# B&R Automation Studio project NAELD004C00R10L518F00 (part 6)

#### Act_Main_P1021.st
```iecst
ACTION Act_Main_P1021:

	//Machine Setting - General
	tyP1021McSetGen.tyGen.tyNumConvInitTm.diValueMin	:= p_tyNtParamCurr.tyUIConvInitTm.diMin;
	tyP1021McSetGen.tyGen.tyNumConvInitTm.diValueMax	:= p_tyNtParamCurr.tyUIConvInitTm.diMax;

	tyP1021McSetGen.tyGen.tyNumMag1ConvRunTm.diValueMin	:= p_tyNtParamCurr.tyUIMagConvRunTm.diMin;
	tyP1021McSetGen.tyGen.tyNumMag1ConvRunTm.diValueMax	:= p_tyNtParamCurr.tyUIMagConvRunTm.diMax;
	tyP1021McSetGen.tyGen.tyNumMag2ConvRunTm.diValueMin	:= p_tyNtParamCurr.tyUIMagConvRunTm.diMin;
	tyP1021McSetGen.tyGen.tyNumMag2ConvRunTm.diValueMax	:= p_tyNtParamCurr.tyUIMagConvRunTm.diMax;
	tyP1021McSetGen.tyGen.tyNumMag3ConvRunTm.diValueMin	:= p_tyNtParamCurr.tyUIMagConvRunTm.diMin;
	tyP1021McSetGen.tyGen.tyNumMag3ConvRunTm.diValueMax	:= p_tyNtParamCurr.tyUIMagConvRunTm.diMax;
	tyP1021McSetGen.tyGen.tyNumMag4ConvRunTm.diValueMin	:= p_tyNtParamCurr.tyUIMagConvRunTm.diMin;
	tyP1021McSetGen.tyGen.tyNumMag4ConvRunTm.diValueMax	:= p_tyNtParamCurr.tyUIMagConvRunTm.diMax;

	tyP1021McSetGen.tyGen.tyNumTranOutErrDlyTm.diValueMin	:= p_tyNtParamCurr.tyUITranOutErrDlyTm.diMin;
	tyP1021McSetGen.tyGen.tyNumTranOutErrDlyTm.diValueMax	:= p_tyNtParamCurr.tyUITranOutErrDlyTm.diMax;

	//LMC feedback time
	tyP1021McSetGen.tyGen.tyNumLMCFbTm.uiRtStat	:= NOT p_tyNtParamCurr.bProjWorkOrderOPCUA;

	//Screen Saver
	tyP1021McSetGen.tyGen.tyNumSSaverTm.diValueMin	:= p_tyNtParamCurr.tyUISSaverTm.diMin;
	tyP1021McSetGen.tyGen.tyNumSSaverTm.diValueMax	:= p_tyNtParamCurr.tyUISSaverTm.diMax;
	tyP1021McSetGen.tyGen.tyNumSSaverTm.uiRtStat.0	:= NOT p_tyNtParamCurr.bSSaverPrep;
	tyP1021McSetGen.tyGen.tyBtnSSaverEn.uiRtStat.0	:= NOT p_tyNtParamCurr.bSSaverPrep;
	tyP1021McSetGen.tyGen.tyTxtLblSSaver.uiRtStat.0	:= NOT p_tyNtParamCurr.bSSaverPrep;

	//Width
	tyP1021McSetGen.tyGen.tyNumWidthAtHm.diValueMin	:= p_tyNtParamCurr.tyProdRcpWidth.diMin;
	tyP1021McSetGen.tyGen.tyNumWidthAtHm.diValueMax	:= p_tyNtParamCurr.tyProdRcpWidth.diMax + 10000;
	tyP1021McSetGen.tyGen.tyNumWidthAtHm.uiRtStat.0	:= NOT p_tyNtParamCurr.bAWPrep;
	tyP1021McSetGen.tyGen.tyTxtWidthAtHm.uiRtStat.0	:= NOT p_tyNtParamCurr.bAWPrep;
	tyP1021McSetGen.tyGen.tyBtnAWDis.uiRtStat.0		:= NOT p_tyNtParamCurr.bAWPrep;

	//Pusher Auto Width AT Home
	tyP1021McSetGen.tyGen.tyNumAWPusherAtHm.diValueMin	:= p_tyNtParamCurr.tyProdRcpWidth.diMin-p_tyNtParamCurr.tyProdRcpWidth.diMin;
	tyP1021McSetGen.tyGen.tyNumAWPusherAtHm.diValueMax	:= (p_tyNtParamCurr.tyProdRcpWidth.diMax + 10000) / 2;
	tyP1021McSetGen.tyGen.tyNumAWPusherAtHm.uiRtStat.0	:= NOT p_tyNtParamCurr.bAWPusherPrep;
	tyP1021McSetGen.tyGen.tyTxtAWPusherAtHm.uiRtStat.0	:= NOT p_tyNtParamCurr.bAWPusherPrep;
	tyP1021McSetGen.tyGen.tyBtnAWPusherDis.uiRtStat.0	:= NOT p_tyNtParamCurr.bAWPusherPrep;

//	tyP1021McSetGen.tyGen.tyNumWidthOffset.uiRtStat.0 :=  NOT p_tyNtParamCurr.bAWPrep;
//	tyP1021McSetGen.tyGen.tyTxtWidthOffset.uiRtStat.0 :=  NOT p_tyNtParamCurr.bAWPrep;
	tyP1021McSetGen.tyGen.tyNumWidthOffset.uiRtStat.0 := TRUE;
	tyP1021McSetGen.tyGen.tyTxtWidthOffset.uiRtStat.0 := TRUE;
	tyP1021McSetGen.tyGen.tyNumWidthOffset.diValueMin :=  p_tyNtParamCurr.tyUIAWOffset.diMin;
	tyP1021McSetGen.tyGen.tyNumWidthOffset.diValueMax :=  p_tyNtParamCurr.tyUIAWOffset.diMax;
	//Hermes Remote Configuration
	tyP1021McSetGen.tyGen.tyBtnHermesRmtEn.uiRtStat.0	:= NOT p_tyNtParamCurr.bHermesRmtPrep;

	//Machine Mode
	tyP1021McSetGen.tyGen.tyDrpDnDefaultMcMod.uiRtStat.0 := TRUE;
	IF p_tyNtParamCurr.bProjLaneBPrep THEN
		tyP1021McSetGen.tyGen.tyDrpDnDefaultMcMod.usiValueMaxIdx	:= 2;
	ELSE
		tyP1021McSetGen.tyGen.tyDrpDnDefaultMcMod.usiValueMaxIdx	:= 0;
	END_IF

	//Flipped Board
	tyP1021McSetGen.tyGen.tyDrpDnDefaultFlippedBrd.usiValueMaxIdx	:= 2;

	//Fix To Fix Rail Machine
	IF p_tyNtParamCurr.bProjLaneBPrep AND p_tyNtParamCurr.bProjDSFixToFixRail THEN
		tyP1021McSetGen.tyGen.tyNumTravFixtoFixPosOutlet.uiRtStat.0 := FALSE;
		tyP1021McSetGen.tyGen.tyNumTravLaneBOffset.uiRtStat.0 := FALSE;
	ELSE
		tyP1021McSetGen.tyGen.tyNumTravFixtoFixPosOutlet.uiRtStat.0 := TRUE;
		tyP1021McSetGen.tyGen.tyNumTravLaneBOffset.uiRtStat.0 := TRUE;
	END_IF

	//Trav & Lifter For Lane B
	tyP1021McSetGen.tyGen.tyNumTravPosLaneA.diValueMin		:= p_tyNtParamCurr.tyUITravTargetPos.diMin;
	tyP1021McSetGen.tyGen.tyNumTravPosLaneA.diValueMax		:= p_tyNtParamCurr.tyUITravTargetPos.diMax;
	tyP1021McSetGen.tyGen.tyNumTravPosLaneB.diValueMin		:= p_tyNtParamCurr.tyUITravTargetPos.diMin;
	tyP1021McSetGen.tyGen.tyNumTravPosLaneB.diValueMax		:= p_tyNtParamCurr.tyUITravTargetPos.diMax;
	tyP1021McSetGen.tyGen.tyNumLiftPosLaneA.diValueMin		:= p_tyNtParamCurr.tyUILifterTargetPos.diMin;
	tyP1021McSetGen.tyGen.tyNumLiftPosLaneA.diValueMax		:= p_tyNtParamCurr.tyUILifterTargetPos.diMax;
	tyP1021McSetGen.tyGen.tyNumLiftPosLaneB.diValueMin		:= p_tyNtParamCurr.tyUILifterTargetPos.diMin;
	tyP1021McSetGen.tyGen.tyNumLiftPosLaneB.diValueMax		:= p_tyNtParamCurr.tyUILifterTargetPos.diMax;
	tyP1021McSetGen.tyGen.tyTxtTravPosLaneB.uiRtStat.0		:= NOT (p_tyNtParamCurr.bProjLaneBPrep AND p_tyNtParamCurr.bProjDSFixToFixRail = FALSE);;
	tyP1021McSetGen.tyGen.tyNumTravPosLaneB.uiRtStat.0		:= NOT (p_tyNtParamCurr.bProjLaneBPrep AND p_tyNtParamCurr.bProjDSFixToFixRail = FALSE);;
	tyP1021McSetGen.tyGen.tyBtnTravPosBTeach.uiRtStat.0		:= NOT (p_tyNtParamCurr.bProjLaneBPrep AND p_tyNtParamCurr.bProjDSFixToFixRail = FALSE);;
	tyP1021McSetGen.tyGen.tyTxtLiftPosLaneB.uiRtStat.0		:= NOT p_tyNtParamCurr.bProjLaneBPrep;
	tyP1021McSetGen.tyGen.tyNumLiftPosLaneB.uiRtStat.0		:= NOT p_tyNtParamCurr.bProjLaneBPrep;
	tyP1021McSetGen.tyGen.tyBtnLiftPosBTeach.uiRtStat.0		:= NOT p_tyNtParamCurr.bProjLaneBPrep;

	//Machine Setting - Magazine Inlet Sensor Auto Detect Timer
	tyP1021McSetGen.tyGen.tyNumMagAutoDetSenTm.diValueMin	:= p_tyNtParamCurr.tyUIMcParamMagAutoEntSenTm.diMin;
	tyP1021McSetGen.tyGen.tyNumMagAutoDetSenTm.diValueMax	:= p_tyNtParamCurr.tyUIMcParamMagAutoEntSenTm.diMax;

	//Vitrual SMEMA
	tyP1021McSetGen.tyGen.tyBtnVSMEMAEn.uiRtStat.0	:= NOT p_tyNtParamCurr.bVSMEMAPrep;

	//Long Board
	tyP1021McSetGen.tyGen.tyBtnLongBrdEn.uiRtStat.0	:= NOT p_tyNtParamCurr.bProjLongBrdPrep;

	//Shutter
	tyP1021McSetGen.tyGen.tyBtnOutShutterDis.uiRtStat.0	:= NOT p_tyNtParamCurr.bProjOutletShutPrep;

	//Magazine Conveyor
	tyP1021McSetGen.tyGen.tyNumMag1ConvRunTm.uiRtStat.0		:= NOT (p_tyNtParamCurr.bProjMag1ConvPrep AND p_tyNtParamCurr.bProjLifTravMnlLoad = FALSE);
	tyP1021McSetGen.tyGen.tyTxtMag1ConvRunTm.uiRtStat.0		:= NOT (p_tyNtParamCurr.bProjMag1ConvPrep AND p_tyNtParamCurr.bProjLifTravMnlLoad = FALSE);
	tyP1021McSetGen.tyGen.tyNumMag2ConvRunTm.uiRtStat.0		:= NOT (p_tyNtParamCurr.bProjMag2ConvPrep AND p_tyNtParamCurr.bProjLifTravMnlLoad = FALSE);
	tyP1021McSetGen.tyGen.tyTxtMag2ConvRunTm.uiRtStat.0		:= NOT (p_tyNtParamCurr.bProjMag2ConvPrep AND p_tyNtParamCurr.bProjLifTravMnlLoad = FALSE);
	tyP1021McSetGen.tyGen.tyNumMag3ConvRunTm.uiRtStat.0		:= NOT(p_tyNtParamCurr.bProjMag3ConvPrep AND (p_tyNtParamCurr.eProjMag = LDMagTriple OR p_tyNtParamCurr.eProjMag = LDMagQuadruple)AND p_tyNtParamCurr.bProjLifTravMnlLoad = FALSE);
	tyP1021McSetGen.tyGen.tyTxtMag3ConvRunTm.uiRtStat.0		:= NOT(p_tyNtParamCurr.bProjMag3ConvPrep AND (p_tyNtParamCurr.eProjMag = LDMagTriple OR p_tyNtParamCurr.eProjMag = LDMagQuadruple)AND p_tyNtParamCurr.bProjLifTravMnlLoad = FALSE);
	tyP1021McSetGen.tyGen.tyNumMag4ConvRunTm.uiRtStat.0		:= NOT(p_tyNtParamCurr.bProjMag4ConvPrep AND (p_tyNtParamCurr.eProjMag = LDMagQuadruple)AND p_tyNtParamCurr.bProjLifTravMnlLoad = FALSE);
	tyP1021McSetGen.tyGen.tyTxtMag4ConvRunTm.uiRtStat.0		:= NOT(p_tyNtParamCurr.bProjMag4ConvPrep AND (p_tyNtParamCurr.eProjMag = LDMagQuadruple)AND p_tyNtParamCurr.bProjLifTravMnlLoad = FALSE);

	//Hermes Supervisory Configuration
	tyP1021McSetGen.tyGen.tyBtnHermesSvyEn.uiRtStat.0		:= NOT p_tyNtParamCurr.bHermesSvyPrep; //new for Hermes 1.3
	tyP1021McSetGen.tyGen.tyBtnRFIDEn.uiRtStat.0			:= NOT (p_tyNtParamCurr.bHermesSvyPrep OR p_tyNtParamCurr.eCustomerReq = We_Fabricate) ;
	tyP1021McSetGen.tyGen.tyNumRFIDWrTO.uiRtStat.0			:= NOT p_tyNtParamCurr.bHermesSvyPrep;

	//Parameter
	tyP1021McSetGen.tyGen.tyStringMcNm.sValue					:= p_tyMcParamCurr.sMcNm;
	tyP1021McSetGen.tyGen.tyDrpDnDefaultMcMod.usiValueIdx		:= p_tyMcParamCurr.usiDefaultMcMod;
	tyP1021McSetGen.tyGen.tyDrpDnDefaultFlippedBrd.usiValueIdx	:= p_tyMcParamCurr.usiDefaultFlippedBrd;
	tyP1021McSetGen.tyGen.tyNumSSaverTm.diValue					:= UINT_TO_DINT(p_tyMcParamCurr.uiSSaverTmInSec);
	tyP1021McSetGen.tyGen.tyBtnSSaverEn.bValue					:= p_tyMcParamCurr.bSSaverEn;
	tyP1021McSetGen.tyGen.tyStringIPAddr.sValue					:= p_sHWInfoIPAddr;
	tyP1021McSetGen.tyGen.tyStringSubnetMask.sValue				:= p_sHWInfoSubnetMask;
	tyP1021McSetGen.tyGen.tyNumWidthAtHm.diValue				:= p_tyMcParamCurr.diWidthAtHmPosInUM;
	tyP1021McSetGen.tyGen.tyNumConvInitTm.diValue				:= p_tyMcParamCurr.diConvInitTmInMS;
	tyP1021McSetGen.tyGen.tyNumTranOutErrDlyTm.diValue			:= p_tyMcParamCurr.diTranOutErrDlyTmInMS;
	tyP1021McSetGen.tyGen.tyNumMag1ConvRunTm.diValue			:= p_tyMcParamCurr.diMag1ConvRunTmOutInMS;
	tyP1021McSetGen.tyGen.tyNumMag2ConvRunTm.diValue			:= p_tyMcParamCurr.diMag2ConvRunTmOutInMS;
	tyP1021McSetGen.tyGen.tyNumMag3ConvRunTm.diValue			:= p_tyMcParamCurr.diMag3ConvRunTmOutInMS;
	tyP1021McSetGen.tyGen.tyNumMag4ConvRunTm.diValue			:= p_tyMcParamCurr.diMag4ConvRunTmOutInMS;
	tyP1021McSetGen.tyGen.tyNumMagAutoDetSenTm.diValue			:= p_tyMcParamCurr.diMagAutoDetectSenTmInMS;

	tyP1021McSetGen.tyGen.tyNumTravPosLaneA.diValue				:= p_tyMcParamCurr.diTravPosA;
	tyP1021McSetGen.tyGen.tyNumLiftPosLaneA.diValue				:= p_tyMcParamCurr.diLifterPosA;
	tyP1021McSetGen.tyGen.tyNumTravPosLaneB.diValue				:= p_tyMcParamCurr.diTravPosB;
	tyP1021McSetGen.tyGen.tyNumLiftPosLaneB.diValue				:= p_tyMcParamCurr.diLifterPosB;

	tyP1021McSetGen.tyGen.tyBtnAWDis.bValue						:= p_tyMcParamCurr.bAWDis;
	tyP1021McSetGen.tyGen.tyBtnAWPusherDis.bValue				:= p_tyMcParamCurr.bAWPusherDis;
	tyP1021McSetGen.tyGen.tyBtnMnlAccDat.bValue					:= p_tyMcParamCurr.bMnlAccDat;
	tyP1021McSetGen.tyGen.tyBtnAutoStepEn.bValue				:= p_tyMcParamCurr.bAutoStepEn;
	tyP1021McSetGen.tyGen.tyBtnVSMEMAEn.bValue					:= p_tyMcParamCurr.bVSMEMAEn;
	tyP1021McSetGen.tyGen.tyBtnHermesRmtEn.bValue				:= p_tyMcParamCurr.bHermesRmtEn;
	tyP1021McSetGen.tyGen.tyBtnLongBrdEn.bValue					:= p_tyMcParamCurr.bLongBrdEn;
	tyP1021McSetGen.tyGen.tyBtnOutShutterDis.bValue				:= p_tyMcParamCurr.bOutShutterDis;
	tyP1021McSetGen.tyGen.tyBtnChgParamEn.bValue				:= p_tyMcParamCurr.bChgParamEn;
	tyP1021McSetGen.tyGen.tyBtnAGVComEn.bValue					:= p_tyMcParamCurr.bAGVComEn;
	tyP1021McSetGen.tyGen.tyNumWidthOffset.diValue				:= p_tyMcParamCurr.diWidthOffsetInUM;

	tyP1021McSetGen.tyGen.tyNumAWPusherAtHm.diValue				:= p_tyMcParamCurr.diAWPusherAtHmPosInUM;

	tyP1021McSetGen.tyGen.tyDrpDnDefaultMcMod.uiRtStat			:= TRUE;
	tyP1021McSetGen.tyGen.tyDrpDnDefaultFlippedBrd.uiRtStat		:= TRUE;
	tyP1021McSetGen.tyGen.tyNumLMCFbTm.diValue 					:= p_tyMcParamCurr.diLMCfbTmInMS;  //LMC fb via opcua
	tyP1021McSetGen.tyGen.tyBtnMagWidthChkDis.bValue 			:= p_tyMcParamCurr.bMagWidthChkDis;
	tyP1021McSetGen.tyGen.tyNumMag1WidthChkDetDist.diValue 		:= p_tyMcParamCurr.diMag1WidthChkDetDist;
	tyP1021McSetGen.tyGen.tyNumMag2WidthChkDetDist.diValue 		:= p_tyMcParamCurr.diMag2WidthChkDetDist;
	tyP1021McSetGen.tyGen.tyNumMag3WidthChkDetDist.diValue 		:= p_tyMcParamCurr.diMag3WidthChkDetDist;

	//Logout
	tyP1021McSetGen.tyGen.tyNumAutoLogoutTm.diValueMin			:= p_tyNtParamCurr.tyUIAutoLogoutTm.diMin;
	tyP1021McSetGen.tyGen.tyNumAutoLogoutTm.diValueMax			:= p_tyNtParamCurr.tyUIAutoLogoutTm.diMax;
	tyP1021McSetGen.tyGen.tyNumAutoLogoutTm.uiRtStat.0			:= NOT p_tyNtParamCurr.bAutoLogoutPrep;
	tyP1021McSetGen.tyGen.tyBtnAutoLogoutEn.uiRtStat.0			:= NOT p_tyNtParamCurr.bAutoLogoutPrep;
	tyP1021McSetGen.tyGen.tyTxtLblAutoLogoutTm.uiRtStat.0		:= NOT p_tyNtParamCurr.bAutoLogoutPrep;

	tyP1021McSetGen.tyGen.tyNumAutoLogoutTm.diValue				:= p_tyMcParamCurr.diAutoLogoutTmInSec;
	tyP1021McSetGen.tyGen.tyBtnAutoLogoutEn.bValue				:= p_tyMcParamCurr.bAutoLogoutEn;

	//Network Mode
	tyP1021McSetGen.tyGen.tyDrpDnNetworkMod.usiValueMinIdx		:= DINT_TO_USINT(p_tyNtParamCurr.tyNetworkMode.diMin);
	tyP1021McSetGen.tyGen.tyDrpDnNetworkMod.usiValueMaxIdx		:= DINT_TO_USINT(p_tyNtParamCurr.tyNetworkMode.diMax);
	tyP1021McSetGen.tyGen.tyDrpDnNetworkMod.usiValueIdx			:= DINT_TO_USINT(p_tyMcParamCurr.eNetworkMod);

	tyP1021McSetGen.tyGen.tyBtnLFBuzMute.bValue					:= p_tyMcParamCurr.bLFBuzMute;

	tyP1021McSetGen.tyGen.tyBtnScannerEn.uiRtStat.0		:= NOT p_tyNtParamCurr.bUSBScannerPrep AND NOT p_tyNtParamCurr.bRS232ScannerPrep;

	tyP1021McSetGen.tyGen.tyDrpDnAGVComProtocol.usiValueMaxIdx		:= 2;
	tyP1021McSetGen.tyGen.tyDrpDnAGVComProtocol.usiValueMinIdx		:= 0;

	CASE  p_tyMcParamCurr.eAGVComProtocol OF
		McSetAGVCommOPCUA:
			tyP1021McSetGen.tyGen.tyDrpDnAGVComProtocol.usiValueIdx :=  0;

		McSetAGVCommHardIO:
			tyP1021McSetGen.tyGen.tyDrpDnAGVComProtocol.usiValueIdx :=  1;

		McSetAGVCommDisabled:
			tyP1021McSetGen.tyGen.tyDrpDnAGVComProtocol.usiValueIdx :=  2;
	END_CASE

	tyP1021McSetGen.tyGen.tyDrpDnMagExchangeMode.usiValueMaxIdx		:= 2;
	tyP1021McSetGen.tyGen.tyDrpDnMagExchangeMode.usiValueMinIdx		:= 0;

	CASE  p_tyMcParamCurr.eMagExMode OF
		McSetMagXcAutoManMode:
			tyP1021McSetGen.tyGen.tyDrpDnMagExchangeMode.usiValueIdx := 0;

		McSetMagXcAutoMode:
			tyP1021McSetGen.tyGen.tyDrpDnMagExchangeMode.usiValueIdx := 1;

		McSetMagXcManMode:
			tyP1021McSetGen.tyGen.tyDrpDnMagExchangeMode.usiValueIdx := 2;
	END_CASE

	tyP1021McSetGen.tyGen.tyDrpDnAGVComProtocol.uiRtStat.0 := NOT p_tyNtParamCurr.bProjAGVPrep;
	tyP1021McSetGen.tyGen.tyDrpDnMagExchangeMode.uiRtStat.0 := NOT p_tyNtParamCurr.bProjAGVPrep;

	tyP1021McSetGen.tyGen.tyBtnAGVSizeDisabled.bValue := p_tyMcParamCurr.bAIVSizeDisabled;
	tyP1021McSetGen.tyGen.tyBtnScannerEn.bValue	:= p_tyMcParamCurr.bScannerEn;

	tyP1021McSetGen.tyGen.tyNumTravFixtoFixPosOutlet.diValue	:= p_tyMcParamCurr.diTravOutletFixtoFixPos;
	tyP1021McSetGen.tyGen.tyNumTravFixtoFixPosOutlet.diValueMax	:= 1500000;

	tyP1021McSetGen.tyGen.tyBtnDisableFMWarning.uiRtStat.0 := NOT(p_tyNtParamCurr.bProjAGVPrep);
	tyP1021McSetGen.tyGen.tyBtnDisableFMWarning.bValue	:= p_tyMcParamCurr.bDisableFMWarning;

	tyP1021McSetGen.tyGen.tyBtnAGVSizeDisabled.uiRtStat.0 := NOT(p_tyNtParamCurr.bProjAGVPrep);

	IF p_tyNtParamCurr.bProjLifterMagPlatform THEN
		tyP1021McSetGen.tyGen.tyTxtLiftPosLaneA.usiValueIdx := 15;
	END_IF

	//DBA on right sensor
	tyP1021McSetGen.tyGen.tyBtnDBAOnRgtSen.bValue := p_tyMcParamCurr.bDBAOnRgtSen;

	//Supervisory + mesRFID
	tyP1021McSetGen.tyGen.tyBtnHermesSvyEn.bValue			:= p_tyMcParamCurr.bHermesSvyEn;//new for Hermes 1.3
	tyP1021McSetGen.tyGen.tyBtnRFIDEn.bValue				:= p_tyMcParamCurr.bMesRFIDEn;
	tyP1021McSetGen.tyGen.tyNumRFIDWrTO.diValue			:= p_tyMcParamCurr.diMesRFIDTOInMS;
	//trav b offset
	tyP1021McSetGen.tyGen.tyNumTravLaneBOffset.diValue		:= p_tyMcParamCurr.diTravLaneBOffset;

END_ACTION
```

#### Act_Main_P1022.st
```iecst
ACTION Act_Main_P1022:

	//Machine Setting - Vertical Communicationm Control
	//Display
	tyP1022McSetVComm.tyVComSel.tyBtnLF.uiRtStat.0				:= NOT p_tyNtParamCurr.bLFPrep;
	tyP1022McSetVComm.tyVComSel.tyBtnLCSLF.uiRtStat.0			:= NOT p_tyNtParamCurr.bLCSLFPrep;
	tyP1022McSetVComm.tyVComSel.tyBtnLCSReqRcp.uiRtStat.0		:= NOT p_tyNtParamCurr.bLCSReqRcpPrep;
	tyP1022McSetVComm.tyVComSel.tyBtnLCSManageRcp.uiRtStat.0	:= NOT p_tyNtParamCurr.bLCSManageRcpPrep;
	tyP1022McSetVComm.tyVComSel.tyBtnLCSLiveDat.uiRtStat.0		:= NOT p_tyNtParamCurr.bLCSLiveDatPrep;

	tyP1022McSetVComm.tyLF.tyBtnLeaderMc.uiRtStat.0			:= NOT p_tyNtParamCurr.bLFUsrSetPrep;
	tyP1022McSetVComm.tyLF.tyBtnDSWidthChkEn.uiRtStat.0		:= NOT p_tyNtParamCurr.bDSWidthChkPrep;

	tyP1022McSetVComm.tyLF.tyBtnDBAOnWOAlign.uiRtStat.0			:= NOT p_tyNtParamCurr.bDSWidthChkPrep;

	//Parameter
	tyP1022McSetVComm.tyVComSel.tyBtnLF.bValue				:= p_tyMcParamCurr.bLFEn;
	tyP1022McSetVComm.tyVComSel.tyBtnLCSLF.bValue			:= p_tyMcParamCurr.bLCSLFEn;
	tyP1022McSetVComm.tyVComSel.tyBtnLCSReqRcp.bValue		:= p_tyMcParamCurr.bLCSReqRcpEn;
	tyP1022McSetVComm.tyVComSel.tyBtnLCSManageRcp.bValue	:= p_tyMcParamCurr.bLCSManageRcpEn;
	tyP1022McSetVComm.tyVComSel.tyBtnLCSLiveDat.bValue		:= p_tyMcParamCurr.bLCSLiveDatEn;

	tyP1022McSetVComm.tyLF.tyBtnLeaderMc.bValue			:= p_tyMcParamCurr.bLFLeaderMc;
	tyP1022McSetVComm.tyLF.tyBtnSectionLdr.bValue		:= p_tyMcParamCurr.bSectionLeader;
	tyP1022McSetVComm.tyLF.tyBtnDSWidthChkEn.bValue		:= p_tyMcParamCurr.bDSWidthChkEn;

	tyP1022McSetVComm.tyLF.tyBtnDBAOnWOAlign.bValue			:= p_tyMcParamCurr.bDBAOnWOAlign;

	//new for Hermes 1.3
	tyP1022McSetVComm.tyVComSvy.tyNumSndAliveTm.diValue	    	    := TIME_TO_DINT(p_tyHermesConfiguration.tySvyParam.tSndAlive);
	tyP1022McSetVComm.tyVComSvy.tyNumSvySystemPort.diValue	    	:= UINT_TO_DINT(p_tyHermesConfiguration.tySvyParam.uiSvySvstemPort);
	tyP1022McSetVComm.tyVComSvy.tyBtnConfiguration.bValue		    := p_tyHermesConfiguration.tySvyParam.bFeatureConfiguration;
	tyP1022McSetVComm.tyVComSvy.tyBtnCheckAliveResponse.bValue		:= p_tyHermesConfiguration.tySvyParam.bFeatureCheckAliveResponse;
	tyP1022McSetVComm.tyVComSvy.tyBtnBoardTracking.bValue		    := p_tyHermesConfiguration.tySvyParam.bFeatureBoardTracking;
	tyP1022McSetVComm.tyVComSvy.tyBtnQueryWorkOrderInfo.bValue		:= p_tyHermesConfiguration.tySvyParam.bFeatureQueryWorkOrderInfo;
	tyP1022McSetVComm.tyVComSvy.tyBtnSendWorkOrderInfo.bValue		:= p_tyHermesConfiguration.tySvyParam.bFeatureSendWorkOrderInfo;

END_ACTION
```

#### Act_Main_P1023.st
```iecst
ACTION Act_Main_P1023:

	//Machine Setting - Horizontal Communicationm Control
	//Display
	tyP1023McSetHComm.tyDSSelA.tyBtnHermes.uiRtStat.0	:= NOT p_tyNtParamCurr.bHermesPrep;
	tyP1023McSetHComm.tyDSSelB.tyBtnHermes.uiRtStat.0	:= NOT p_tyNtParamCurr.bHermesPrep;

	tyP1023McSetHComm.tyDSHermesA.tyBtnBoardForecast.uiRtStat.0	:= NOT p_tyNtParamCurr.bHermesSvyPrep;
	tyP1023McSetHComm.tyDSHermesA.tyBtnSendBoardInfo.uiRtStat.0	:= NOT p_tyNtParamCurr.bHermesSvyPrep;

	IF p_tyNtParamCurr.bIPCSMEMA9851ExtdPrep = TRUE THEN
		tyP1023McSetHComm.tyDSSMEMAA.tyDrpDnSMEMAMod.usiValueMaxIdx	:= 2;
		tyP1023McSetHComm.tyDSSMEMAB.tyDrpDnSMEMAMod.usiValueMaxIdx	:= 2;
	ELSE
		tyP1023McSetHComm.tyDSSMEMAA.tyDrpDnSMEMAMod.usiValueMaxIdx	:= 1;
		tyP1023McSetHComm.tyDSSMEMAB.tyDrpDnSMEMAMod.usiValueMaxIdx	:= 1;
	END_IF

	tyP1023McSetHComm.tyDSHermesA.tyNumSndAliveTm.diValueMin	:= p_tyNtParamCurr.tyUIHermesSndAliveTm.diMin;
	tyP1023McSetHComm.tyDSHermesA.tyNumSndAliveTm.diValueMax	:= p_tyNtParamCurr.tyUIHermesSndAliveTm.diMax;
	tyP1023McSetHComm.tyDSHermesB.tyNumSndAliveTm.diValueMin	:= p_tyNtParamCurr.tyUIHermesSndAliveTm.diMin;
	tyP1023McSetHComm.tyDSHermesB.tyNumSndAliveTm.diValueMax	:= p_tyNtParamCurr.tyUIHermesSndAliveTm.diMax;

	tyP1023McSetHComm.tyDSHermesA.tyNumLaneID.diValueMin		:= p_tyNtParamCurr.tyUIHermesLnID.diMin;
	tyP1023McSetHComm.tyDSHermesA.tyNumLaneID.diValueMax		:= p_tyNtParamCurr.tyUIHermesLnID.diMax;
	tyP1023McSetHComm.tyDSHermesB.tyNumLaneID.diValueMin		:= p_tyNtParamCurr.tyUIHermesLnID.diMin;
	tyP1023McSetHComm.tyDSHermesB.tyNumLaneID.diValueMax		:= p_tyNtParamCurr.tyUIHermesLnID.diMax;

	//Parameter - Downstream A
	CASE p_tyMcParamCurr.eDSCommA OF
		McSetCommModSMEMA:
			tyP1023McSetHComm.tyDSSelA.tyBtnSMEMA.bValue	:= TRUE;
			tyP1023McSetHComm.tyDSSelA.tyBtnSMEMA.bRtLk		:= TRUE;
			tyP1023McSetHComm.tyDSSelA.tyBtnHermes.bValue	:= FALSE;
			tyP1023McSetHComm.tyDSSelA.tyBtnHermes.bRtLk	:= FALSE;
		McSetCommModHermes:
			tyP1023McSetHComm.tyDSSelA.tyBtnSMEMA.bValue	:= FALSE;
			tyP1023McSetHComm.tyDSSelA.tyBtnSMEMA.bRtLk		:= FALSE;
			tyP1023McSetHComm.tyDSSelA.tyBtnHermes.bValue	:= TRUE;
			tyP1023McSetHComm.tyDSSelA.tyBtnHermes.bRtLk	:= TRUE;
	END_CASE

	tyP1023McSetHComm.tyDSSMEMAA.tyDrpDnSMEMAMod.usiValueIdx		:= UDINT_TO_USINT(p_tyMcParamCurr.tyDSCommASMEMA.eSelection);
	tyP1023McSetHComm.tyDSSMEMAA.tyBtnGdSig.bValue					:= p_tyMcParamCurr.tyDSCommASMEMA.bStatSigSetGd;

	tyP1023McSetHComm.tyDSHermesA.tyNumSndAliveTm.diValue			:= TIME_TO_DINT(p_tyHermesConfiguration.a_tyDSParam[0].tSndAlive);
	tyP1023McSetHComm.tyDSHermesA.tyNumSvrPort.diValue				:= UINT_TO_DINT(p_tyHermesConfiguration.a_tyDSParam[0].uiSvrPort);
	tyP1023McSetHComm.tyDSHermesA.tyNumLaneID.diValue				:= INT_TO_DINT(p_tyHermesConfiguration.a_tyDSParam[0].iLaneID);
	tyP1023McSetHComm.tyDSHermesA.tyBtnCheckAliveResponse.bValue	:= p_tyHermesConfiguration.a_tyDSParam[0].bFeatureCheckAliveResponse;
	tyP1023McSetHComm.tyDSHermesA.tyBtnBoardForecast.bValue	:= p_tyHermesConfiguration.a_tyDSParam[0].bFeatureBoardForecast;//new for Hermes 1.3
	tyP1023McSetHComm.tyDSHermesA.tyBtnSendBoardInfo.bValue	:= p_tyHermesConfiguration.a_tyDSParam[0].bFeatureSendBoardInfo;//new for Hermes 1.3

	//Parameter - Downstream B
	CASE p_tyMcParamCurr.eDSCommB OF
		McSetCommModSMEMA:
			tyP1023McSetHComm.tyDSSelB.tyBtnSMEMA.bValue	:= TRUE;
			tyP1023McSetHComm.tyDSSelB.tyBtnSMEMA.bRtLk		:= TRUE;
			tyP1023McSetHComm.tyDSSelB.tyBtnHermes.bValue	:= FALSE;
			tyP1023McSetHComm.tyDSSelB.tyBtnHermes.bRtLk	:= FALSE;
		McSetCommModHermes:
			tyP1023McSetHComm.tyDSSelB.tyBtnSMEMA.bValue	:= FALSE;
			tyP1023McSetHComm.tyDSSelB.tyBtnSMEMA.bRtLk		:= FALSE;
			tyP1023McSetHComm.tyDSSelB.tyBtnHermes.bValue	:= TRUE;
			tyP1023McSetHComm.tyDSSelB.tyBtnHermes.bRtLk	:= TRUE;
	END_CASE

	tyP1023McSetHComm.tyDSSMEMAB.tyDrpDnSMEMAMod.usiValueIdx		:= UDINT_TO_USINT(p_tyMcParamCurr.tyDSCommBSMEMA.eSelection);
	tyP1023McSetHComm.tyDSSMEMAB.tyBtnGdSig.bValue					:= p_tyMcParamCurr.tyDSCommBSMEMA.bStatSigSetGd;

	tyP1023McSetHComm.tyDSHermesB.tyNumSndAliveTm.diValue			:= TIME_TO_DINT(p_tyHermesConfiguration.a_tyDSParam[1].tSndAlive);
	tyP1023McSetHComm.tyDSHermesB.tyNumSvrPort.diValue				:= UINT_TO_DINT(p_tyHermesConfiguration.a_tyDSParam[1].uiSvrPort);
	tyP1023McSetHComm.tyDSHermesB.tyNumLaneID.diValue				:= INT_TO_DINT(p_tyHermesConfiguration.a_tyDSParam[1].iLaneID);
	tyP1023McSetHComm.tyDSHermesB.tyBtnCheckAliveResponse.bValue	:= p_tyHermesConfiguration.a_tyDSParam[1].bFeatureCheckAliveResponse;
	tyP1023McSetHComm.tyDSHermesB.tyBtnBoardForecast.bValue	:= p_tyHermesConfiguration.a_tyDSParam[1].bFeatureBoardForecast;//new for Hermes 1.3
	tyP1023McSetHComm.tyDSHermesB.tyBtnSendBoardInfo.bValue	:= p_tyHermesConfiguration.a_tyDSParam[1].bFeatureSendBoardInfo;//new for Hermes 1.3

END_ACTION
```

#### Act_Main_P1024.st
```iecst
ACTION Act_Main_P1024:

	//Machine Setting - Anti Gap Sensor Filter
	tyP1024McSetAntiGap.tyAntiGap.tyNumLftSenOff.diValueMin	:= p_tyNtParamCurr.tyUIAntiGapSenOffTm.diMin;
	tyP1024McSetAntiGap.tyAntiGap.tyNumLftSenOff.diValueMax	:= p_tyNtParamCurr.tyUIAntiGapSenOffTm.diMax;

	tyP1024McSetAntiGap.tyAntiGap.tyNumRgtSenOff.diValueMin	:= p_tyNtParamCurr.tyUIAntiGapSenOffTm.diMin;
	tyP1024McSetAntiGap.tyAntiGap.tyNumRgtSenOff.diValueMax	:= p_tyNtParamCurr.tyUIAntiGapSenOffTm.diMax;

	tyP1024McSetAntiGap.tyAntiGap.tyNumMagConvEntOff.diValueMin	:= p_tyNtParamCurr.tyUIAntiGapSenOffTm.diMin;
	tyP1024McSetAntiGap.tyAntiGap.tyNumMagConvEntOff.diValueMax	:= p_tyNtParamCurr.tyUIAntiGapSenOffTm.diMax;

	tyP1024McSetAntiGap.tyAntiGap.tyNumMagConvEntOn.diValueMin	:= p_tyNtParamCurr.tyUIAntiGapSenOnTm.diMin;
	tyP1024McSetAntiGap.tyAntiGap.tyNumMagConvEntOn.diValueMax	:= p_tyNtParamCurr.tyUIAntiGapSenOnTm.diMax;

	tyP1024McSetAntiGap.tyAntiGap.tyNumMagConvPresentOff.diValueMin	:= p_tyNtParamCurr.tyUIAntiGapSenOffTm.diMin;
	tyP1024McSetAntiGap.tyAntiGap.tyNumMagConvPresentOff.diValueMax	:= p_tyNtParamCurr.tyUIAntiGapSenOffTm.diMax;

	tyP1024McSetAntiGap.tyAntiGap.tyNumMagConvPresentOn.diValueMin	:= p_tyNtParamCurr.tyUIAntiGapSenOnTm.diMin;
	tyP1024McSetAntiGap.tyAntiGap.tyNumMagConvPresentOn.diValueMax	:= p_tyNtParamCurr.tyUIAntiGapSenOnTm.diMax;

	//Parameter
	tyP1024McSetAntiGap.tyAntiGap.tyNumLftSenOff.diValue	:= p_tyMcParamCurr.tyLftSenAntiGapDly.diSigOffTm;

	tyP1024McSetAntiGap.tyAntiGap.tyNumRgtSenOff.diValue	:= p_tyMcParamCurr.tyRgtSenAntiGapDly.diSigOffTm;

	tyP1024McSetAntiGap.tyAntiGap.tyNumMagConvEntOff.diValue	:= p_tyMcParamCurr.tyMagConvEntrySenAntiGapDly.diSigOffTm;
	tyP1024McSetAntiGap.tyAntiGap.tyNumMagConvEntOn.diValue		:= p_tyMcParamCurr.tyMagConvEntrySenAntiGapDly.diSigOnTm;

	tyP1024McSetAntiGap.tyAntiGap.tyNumMagConvPresentOff.diValue	:= p_tyMcParamCurr.tyMagConvPresentSenAntiGapDly.diSigOffTm;
	tyP1024McSetAntiGap.tyAntiGap.tyNumMagConvPresentOn.diValue		:= p_tyMcParamCurr.tyMagConvPresentSenAntiGapDly.diSigOnTm;

	tyP1024McSetAntiGap.tyAntiGap.tyNumMagConvEntOff.uiRtStat.0 := NOT (p_tyNtParamCurr.bProjMag1ConvPrep AND p_tyNtParamCurr.bProjMag2ConvPrep AND p_tyNtParamCurr.bProjMag3ConvPrep AND p_tyNtParamCurr.bProjLifTravMnlLoad= FALSE);
	tyP1024McSetAntiGap.tyAntiGap.tyNumMagConvEntOn.uiRtStat.0 := NOT (p_tyNtParamCurr.bProjMag1ConvPrep AND p_tyNtParamCurr.bProjMag2ConvPrep AND p_tyNtParamCurr.bProjMag3ConvPrep AND p_tyNtParamCurr.bProjLifTravMnlLoad= FALSE);
	tyP1024McSetAntiGap.tyAntiGap.tyNumMagConvPresentOff.uiRtStat.0 := NOT (p_tyNtParamCurr.bProjMag1ConvPrep AND p_tyNtParamCurr.bProjMag2ConvPrep AND p_tyNtParamCurr.bProjMag3ConvPrep);
	tyP1024McSetAntiGap.tyAntiGap.tyNumMagConvPresentOn.uiRtStat.0 := NOT (p_tyNtParamCurr.bProjMag1ConvPrep AND p_tyNtParamCurr.bProjMag2ConvPrep AND p_tyNtParamCurr.bProjMag3ConvPrep);

END_ACTION
```

#### Act_Main_P1025.st
```iecst
ACTION Act_Main_P1025:

	//Machine Setting - AIV Communication
	//Parameter
//	tyP1025McSetAIVComm.tyAIVComm.tyNumSvrPort.diValue		:= UINT_TO_DINT(p_tyMcParamCurr.tyAIVComm.uiSvrPort);
//	tyP1025McSetAIVComm.tyAIVComm.tyNumAllwClntPort.diValue	:= UINT_TO_DINT(p_tyMcParamCurr.tyAIVComm.uiClientPort);
//	tyP1025McSetAIVComm.tyAIVComm.tyStringAllwClntIP.sValue	:= p_tyMcParamCurr.tyAIVComm.sClientAddress;

END_ACTION
```

#### Act_Main_P1026.st
```iecst
ACTION Act_Main_P1026:

	//Display
	//Curtain sensor bypass
	IF p_tyNtParamCurr.tyDOSettings.diBypCurtainSen > 0 THEN
		tyP1026McSetTeach.tyTeachLifterPosA.tyBtn4.uiRtStat := FALSE;
		tyP1026McSetTeach.tyTeachLifterPosA.tyBtn4.usiBitmapIdx := 5;
		tyP1026McSetTeach.tyTeachLifterPosA.tyBtn4.usiTxtIdx := 47;
		tyP1026McSetTeach.tyTeachLifterPosB.tyBtn4.uiRtStat := FALSE;
		tyP1026McSetTeach.tyTeachLifterPosB.tyBtn4.usiBitmapIdx := 5;
		tyP1026McSetTeach.tyTeachLifterPosB.tyBtn4.usiTxtIdx := 47;
		tyP1026McSetTeach.tyTeachTravPosA.tyBtn4.uiRtStat := FALSE;
		tyP1026McSetTeach.tyTeachTravPosA.tyBtn4.usiBitmapIdx := 5;
		tyP1026McSetTeach.tyTeachTravPosA.tyBtn4.usiTxtIdx := 47;
		tyP1026McSetTeach.tyTeachTravPosB.tyBtn4.uiRtStat := FALSE;
		tyP1026McSetTeach.tyTeachTravPosB.tyBtn4.usiBitmapIdx := 5;
		tyP1026McSetTeach.tyTeachTravPosB.tyBtn4.usiTxtIdx := 47;
	END_IF

	//Traverser
	tyP1026McSetTeach.tyMotionStdTrav.tyNumTargetPos.diValue	:= 0;
	tyP1026McSetTeach.tyMotionStdTrav.tyNumStepSize.diValue		:= 0;
	tyP1026McSetTeach.tyMotionStdTrav.tyNumNomSpd.diValue		:= (p_tyNtParamCurr.tyUITravNomSpd.diMax + p_tyNtParamCurr.tyUITravNomSpd.diMin) / 2;
	tyP1026McSetTeach.tyMotionStdTrav.tyNumSlwSpd.diValue		:= (p_tyNtParamCurr.tyUITravSlwSpd.diMax + p_tyNtParamCurr.tyUITravSlwSpd.diMin) / 3;

	tyP1026McSetTeach.tyMotionStdTrav.tyNumTargetPos.diValueMax	:= p_tyNtParamCurr.tyUITravTargetPos.diMax;
	tyP1026McSetTeach.tyMotionStdTrav.tyNumTargetPos.diValueMin	:= p_tyNtParamCurr.tyUITravTargetPos.diMin;

	tyP1026McSetTeach.tyMotionStdTrav.tyNumStepSize.diValueMax	:= p_tyNtParamCurr.tyUITravStepSize.diMax;
	tyP1026McSetTeach.tyMotionStdTrav.tyNumStepSize.diValueMin	:= p_tyNtParamCurr.tyUITravStepSize.diMin;

	tyP1026McSetTeach.tyMotionStdTrav.tyNumNomSpd.diValueMax	:= p_tyNtParamCurr.tyUITravNomSpd.diMax;
	tyP1026McSetTeach.tyMotionStdTrav.tyNumNomSpd.diValueMin	:= p_tyNtParamCurr.tyUITravNomSpd.diMin;

	tyP1026McSetTeach.tyMotionStdTrav.tyNumSlwSpd.diValueMax	:= p_tyNtParamCurr.tyUITravSlwSpd.diMax;
	tyP1026McSetTeach.tyMotionStdTrav.tyNumSlwSpd.diValueMin	:= p_tyNtParamCurr.tyUITravSlwSpd.diMin;

	//Lifter
	tyP1026McSetTeach.tyMotionStdLifter.tyNumTargetPos.diValue		:= 0;
	tyP1026McSetTeach.tyMotionStdLifter.tyNumStepSize.diValue		:= 0;
	tyP1026McSetTeach.tyMotionStdLifter.tyNumNomSpd.diValue			:= (p_tyNtParamCurr.tyUILifterNomSpd.diMax + p_tyNtParamCurr.tyUILifterNomSpd.diMin) / 2;
	tyP1026McSetTeach.tyMotionStdLifter.tyNumSlwSpd.diValue			:= (p_tyNtParamCurr.tyUILifterSlwSpd.diMax + p_tyNtParamCurr.tyUILifterSlwSpd.diMin) / 3;

	tyP1026McSetTeach.tyMotionStdLifter.tyNumTargetPos.diValueMax	:= p_tyNtParamCurr.tyUILifterTargetPos.diMax;
	tyP1026McSetTeach.tyMotionStdLifter.tyNumTargetPos.diValueMin	:= p_tyNtParamCurr.tyUILifterTargetPos.diMin;

	tyP1026McSetTeach.tyMotionStdLifter.tyNumStepSize.diValueMax	:= p_tyNtParamCurr.tyUILifterStepSize.diMax;
	tyP1026McSetTeach.tyMotionStdLifter.tyNumStepSize.diValueMin	:= p_tyNtParamCurr.tyUILifterStepSize.diMin;

	tyP1026McSetTeach.tyMotionStdLifter.tyNumNomSpd.diValueMax		:= p_tyNtParamCurr.tyUILifterNomSpd.diMax;
	tyP1026McSetTeach.tyMotionStdLifter.tyNumNomSpd.diValueMin		:= p_tyNtParamCurr.tyUILifterNomSpd.diMin;

	tyP1026McSetTeach.tyMotionStdLifter.tyNumSlwSpd.diValueMax		:= p_tyNtParamCurr.tyUILifterSlwSpd.diMax;
	tyP1026McSetTeach.tyMotionStdLifter.tyNumSlwSpd.diValueMin		:= p_tyNtParamCurr.tyUILifterSlwSpd.diMin;

END_ACTION
```

#### Act_Main_P1027.st
```iecst
(** 2021-08-20 **)
ACTION Act_Main_P1027:

	tyP1027McSetUSBSetting.tyUSBSet.tyVID.diValue			:= p_tyMcParamCurr.diVID;
	tyP1027McSetUSBSetting.tyUSBSet.tyPID.diValue			:= p_tyMcParamCurr.diPID;

	tyP1027McSetUSBSetting.tyUSBSet.tyVID.diValueMax		:= p_tyNtParamCurr.tyVID.diMax;
	tyP1027McSetUSBSetting.tyUSBSet.tyVID.diValueMin		:= p_tyNtParamCurr.tyVID.diMin;
	tyP1027McSetUSBSetting.tyUSBSet.tyPID.diValueMax		:= p_tyNtParamCurr.tyPID.diMax;
	tyP1027McSetUSBSetting.tyUSBSet.tyPID.diValueMin		:= p_tyNtParamCurr.tyPID.diMin;

END_ACTION
```

#### Act_Main_P1028.st
```iecst
(** 2021-08-20 **)
ACTION Act_Main_P1028:

	//Parameter
	tyP1028McSetRS232Setting.tyRS232Set.tyNumStartCode1.diValue	:= p_tyMcParamCurr.diRS232StartCode1;
	tyP1028McSetRS232Setting.tyRS232Set.tyNumStartCode2.diValue	:= p_tyMcParamCurr.diRS232StartCode2;
	tyP1028McSetRS232Setting.tyRS232Set.tyNumEndCode1.diValue	:= p_tyMcParamCurr.diRS232EndCode1;
	tyP1028McSetRS232Setting.tyRS232Set.tyNumEndCode2.diValue	:= p_tyMcParamCurr.diRS232EndCode2;

END_ACTION
```

#### Act_Main_P1030.st
```iecst
ACTION Act_Main_P1030:

	//P1030 Magazine Settings
	//Display
	tyP1030MagSet.tyMagSet.tyTxtLifMag3Slt1PosLbl.uiRtStat.0	:= NOT(p_tyNtParamCurr.eProjMag = LDMagTriple OR p_tyNtParamCurr.eProjMag = LDMagQuadruple);
	tyP1030MagSet.tyMagSet.tyNumLifterMag3Slt1Pos.uiRtStat.0	:= NOT(p_tyNtParamCurr.eProjMag = LDMagTriple OR p_tyNtParamCurr.eProjMag = LDMagQuadruple);
	tyP1030MagSet.tyMagSet.tyBtnLifterMag3Slt1Pos.uiRtStat.0	:= NOT(p_tyNtParamCurr.eProjMag = LDMagTriple OR p_tyNtParamCurr.eProjMag = LDMagQuadruple);

	tyP1030MagSet.tyMagSet.tyTxtTravPosMag3Lbl.uiRtStat.0	:= NOT(p_tyNtParamCurr.eProjMag = LDMagTriple OR p_tyNtParamCurr.eProjMag = LDMagQuadruple);
	tyP1030MagSet.tyMagSet.tyNumTravPosMag3.uiRtStat.0		:= NOT(p_tyNtParamCurr.eProjMag = LDMagTriple OR p_tyNtParamCurr.eProjMag = LDMagQuadruple);
	tyP1030MagSet.tyMagSet.tyBtnTravPosMag3.uiRtStat.0		:= NOT(p_tyNtParamCurr.eProjMag = LDMagTriple OR p_tyNtParamCurr.eProjMag = LDMagQuadruple);

	tyP1030MagSet.tyMagSet.tyNumSltToSltDist.diValueMin	:= p_tyNtParamCurr.tyUISltToSltDist.diMin;
	tyP1030MagSet.tyMagSet.tyNumSltToSltDist.diValueMax	:= p_tyNtParamCurr.tyUISltToSltDist.diMax;

	tyP1030MagSet.tyMagSet.tyNumMaxSlt.diValueMin	:= p_tyNtParamCurr.diProjMagMinSlt;
	tyP1030MagSet.tyMagSet.tyNumMaxSlt.diValueMax	:= p_tyNtParamCurr.diProjMagMaxSlt;

	tyP1030MagSet.tyMagSet.tyNumLifterMag1Slt1Pos.diValueMin	:= p_tyNtParamCurr.tyUILifterTargetPos.diMin;
	tyP1030MagSet.tyMagSet.tyNumLifterMag1Slt1Pos.diValueMax	:= p_tyNtParamCurr.tyUILifterTargetPos.diMax;
	tyP1030MagSet.tyMagSet.tyNumLifterMag2Slt1Pos.diValueMin	:= p_tyNtParamCurr.tyUILifterTargetPos.diMin;
	tyP1030MagSet.tyMagSet.tyNumLifterMag2Slt1Pos.diValueMax	:= p_tyNtParamCurr.tyUILifterTargetPos.diMax;
	tyP1030MagSet.tyMagSet.tyNumLifterMag3Slt1Pos.diValueMin	:= p_tyNtParamCurr.tyUILifterTargetPos.diMin;
	tyP1030MagSet.tyMagSet.tyNumLifterMag3Slt1Pos.diValueMax	:= p_tyNtParamCurr.tyUILifterTargetPos.diMax;

	tyP1030MagSet.tyMagSet.tyNumTravPosMag1.diValueMin	:= p_tyNtParamCurr.tyUITravTargetPos.diMin;
	tyP1030MagSet.tyMagSet.tyNumTravPosMag1.diValueMax	:= p_tyNtParamCurr.tyUITravTargetPos.diMax;
	tyP1030MagSet.tyMagSet.tyNumTravPosMag2.diValueMin	:= p_tyNtParamCurr.tyUITravTargetPos.diMin;
	tyP1030MagSet.tyMagSet.tyNumTravPosMag2.diValueMax	:= p_tyNtParamCurr.tyUITravTargetPos.diMax;
	tyP1030MagSet.tyMagSet.tyNumTravPosMag3.diValueMin	:= p_tyNtParamCurr.tyUITravTargetPos.diMin;
	tyP1030MagSet.tyMagSet.tyNumTravPosMag3.diValueMax	:= p_tyNtParamCurr.tyUITravTargetPos.diMax;
	tyP1030MagSet.tyMagSet.tyNumTravPosMag4.diValueMin	:= p_tyNtParamCurr.tyUITravTargetPos.diMin;
	tyP1030MagSet.tyMagSet.tyNumTravPosMag4.diValueMax	:= p_tyNtParamCurr.tyUITravTargetPos.diMax;

	FOR i := 1 TO c_uiP1030TableSize DO
		tyP1030MagSet.tyMagSet.tyTableRecipe.a_tyStringDataCol0[i].sValue	:= UINT_TO_STRING(i);
		tyP1030MagSet.tyMagSet.tyTableRecipe.a_tyStringDataCol1[i].sValue	:= p_tyMagRcpCurrList[i].sRcpNm;
		tyP1030MagSet.tyMagSet.tyTableRecipe.a_tyStringDataCol2[i].sValue	:= p_tyMagRcpCurrList[i].sDisplayInfo;
	END_FOR

	tyP1030MagSet.tyMagSet.tyDrpDnMagModel.usiValueMaxIdx	:= 2;

	tyP1030MagSet.tyMagSet.tyTxtLifMag4Slt1PosLbl.uiRtStat.0	:= NOT(p_tyNtParamCurr.eProjMag = LDMagQuadruple);
	tyP1030MagSet.tyMagSet.tyNumLifterMag4Slt1Pos.uiRtStat.0	:= NOT(p_tyNtParamCurr.eProjMag = LDMagQuadruple);
	tyP1030MagSet.tyMagSet.tyBtnLifterMag4Slt1Pos.uiRtStat.0	:= NOT(p_tyNtParamCurr.eProjMag = LDMagQuadruple);

	tyP1030MagSet.tyMagSet.tyTxtTravPosMag4Lbl.uiRtStat.0	:= NOT(p_tyNtParamCurr.eProjMag = LDMagQuadruple);
	tyP1030MagSet.tyMagSet.tyNumTravPosMag4.uiRtStat.0		:= NOT( p_tyNtParamCurr.eProjMag = LDMagQuadruple);
	tyP1030MagSet.tyMagSet.tyBtnTravPosMag4.uiRtStat.0		:= NOT(p_tyNtParamCurr.eProjMag = LDMagQuadruple);

	tyP1030MagSet.tyMagSet.tyNumMagMaxBrdWidth.diValueMin		:= p_tyNtParamCurr.tyProdRcpWidth.diMin;
	tyP1030MagSet.tyMagSet.tyNumMagMaxBrdWidth.diValueMax		:= p_tyNtParamCurr.tyProdRcpWidth.diMax;

	tyP1030MagSet.tyMagSet.tyBtnSafetyBarDisabled.uiRtStat.0	:= NOT(p_tyNtParamCurr.bProjMagSafetyBarPrep);
	tyP1030MagSet.tyMagSet.tyBtnMagHeightChkEn.uiRtStat.0	 := NOT(p_tyNtParamCurr.bProjMagHeightChkPrep);
	tyP1030MagSet.tyMagSet.tyBitmapBrder.uiRtStat.0 		 := NOT(p_tyNtParamCurr.bProjMagSafetyBarPrep OR p_tyNtParamCurr.bProjMagHeightChkPrep);

END_ACTION
```

#### Act_Main_P1031.st
```iecst
ACTION Act_Main_P1031:

	//Display
	//Curtain sensor bypass
	IF p_tyNtParamCurr.tyDOSettings.diBypCurtainSen > 0 THEN
		tyP1031MagSetTeach.tyTeachTravPosMag1.tyBtn4.uiRtStat := FALSE;
		tyP1031MagSetTeach.tyTeachTravPosMag1.tyBtn4.usiBitmapIdx := 5;
		tyP1031MagSetTeach.tyTeachTravPosMag1.tyBtn4.usiTxtIdx := 47;
		tyP1031MagSetTeach.tyTeachTravPosMag2.tyBtn4.uiRtStat := FALSE;
		tyP1031MagSetTeach.tyTeachTravPosMag2.tyBtn4.usiBitmapIdx := 5;
		tyP1031MagSetTeach.tyTeachTravPosMag2.tyBtn4.usiTxtIdx := 47;
		tyP1031MagSetTeach.tyTeachTravPosMag3.tyBtn4.uiRtStat := FALSE;
		tyP1031MagSetTeach.tyTeachTravPosMag3.tyBtn4.usiBitmapIdx := 5;
		tyP1031MagSetTeach.tyTeachTravPosMag3.tyBtn4.usiTxtIdx := 47;
		tyP1031MagSetTeach.tyTeachLifterMag1Slt1Pos.tyBtn4.uiRtStat := FALSE;
		tyP1031MagSetTeach.tyTeachLifterMag1Slt1Pos.tyBtn4.usiBitmapIdx := 5;
		tyP1031MagSetTeach.tyTeachLifterMag1Slt1Pos.tyBtn4.usiTxtIdx := 47;
		tyP1031MagSetTeach.tyTeachLifterMag2Slt1Pos.tyBtn4.uiRtStat := FALSE;
		tyP1031MagSetTeach.tyTeachLifterMag2Slt1Pos.tyBtn4.usiBitmapIdx := 5;
		tyP1031MagSetTeach.tyTeachLifterMag2Slt1Pos.tyBtn4.usiTxtIdx := 47;
		tyP1031MagSetTeach.tyTeachLifterMag3Slt1Pos.tyBtn4.uiRtStat := FALSE;
		tyP1031MagSetTeach.tyTeachLifterMag3Slt1Pos.tyBtn4.usiBitmapIdx := 5;
		tyP1031MagSetTeach.tyTeachLifterMag3Slt1Pos.tyBtn4.usiTxtIdx := 47;
	END_IF

	//Traverser
	tyP1031MagSetTeach.tyMotionStdTrav.tyNumTargetPos.diValue		:= 0;
	tyP1031MagSetTeach.tyMotionStdTrav.tyNumStepSize.diValue		:= 0;
	tyP1031MagSetTeach.tyMotionStdTrav.tyNumNomSpd.diValue			:= (p_tyNtParamCurr.tyUITravNomSpd.diMax + p_tyNtParamCurr.tyUITravNomSpd.diMin) / 2;
	tyP1031MagSetTeach.tyMotionStdTrav.tyNumSlwSpd.diValue			:= (p_tyNtParamCurr.tyUITravSlwSpd.diMax + p_tyNtParamCurr.tyUITravSlwSpd.diMin) / 3;

	tyP1031MagSetTeach.tyMotionStdTrav.tyNumTargetPos.diValueMax	:= p_tyNtParamCurr.tyUITravTargetPos.diMax;
	tyP1031MagSetTeach.tyMotionStdTrav.tyNumTargetPos.diValueMin	:= p_tyNtParamCurr.tyUITravTargetPos.diMin;

	tyP1031MagSetTeach.tyMotionStdTrav.tyNumStepSize.diValueMax		:= p_tyNtParamCurr.tyUITravStepSize.diMax;
	tyP1031MagSetTeach.tyMotionStdTrav.tyNumStepSize.diValueMin		:= p_tyNtParamCurr.tyUITravStepSize.diMin;

	tyP1031MagSetTeach.tyMotionStdTrav.tyNumNomSpd.diValueMax		:= p_tyNtParamCurr.tyUITravNomSpd.diMax;
	tyP1031MagSetTeach.tyMotionStdTrav.tyNumNomSpd.diValueMin		:= p_tyNtParamCurr.tyUITravNomSpd.diMin;

	tyP1031MagSetTeach.tyMotionStdTrav.tyNumSlwSpd.diValueMax		:= p_tyNtParamCurr.tyUITravSlwSpd.diMax;
	tyP1031MagSetTeach.tyMotionStdTrav.tyNumSlwSpd.diValueMin		:= p_tyNtParamCurr.tyUITravSlwSpd.diMin;

	//Lifter
	tyP1031MagSetTeach.tyMotionStdLifter.tyNumTargetPos.diValue		:= 0;
	tyP1031MagSetTeach.tyMotionStdLifter.tyNumStepSize.diValue		:= 0;
	tyP1031MagSetTeach.tyMotionStdLifter.tyNumNomSpd.diValue		:= (p_tyNtParamCurr.tyUILifterNomSpd.diMax + p_tyNtParamCurr.tyUILifterNomSpd.diMin) / 2;
	tyP1031MagSetTeach.tyMotionStdLifter.tyNumSlwSpd.diValue		:= (p_tyNtParamCurr.tyUILifterSlwSpd.diMax + p_tyNtParamCurr.tyUILifterSlwSpd.diMin) / 3;

	tyP1031MagSetTeach.tyMotionStdLifter.tyNumTargetPos.diValueMax	:= p_tyNtParamCurr.tyUILifterTargetPos.diMax;
	tyP1031MagSetTeach.tyMotionStdLifter.tyNumTargetPos.diValueMin	:= p_tyNtParamCurr.tyUILifterTargetPos.diMin;

	tyP1031MagSetTeach.tyMotionStdLifter.tyNumStepSize.diValueMax	:= p_tyNtParamCurr.tyUILifterStepSize.diMax;
	tyP1031MagSetTeach.tyMotionStdLifter.tyNumStepSize.diValueMin	:= p_tyNtParamCurr.tyUILifterStepSize.diMin;

	tyP1031MagSetTeach.tyMotionStdLifter.tyNumNomSpd.diValueMax		:= p_tyNtParamCurr.tyUILifterNomSpd.diMax;
	tyP1031MagSetTeach.tyMotionStdLifter.tyNumNomSpd.diValueMin		:= p_tyNtParamCurr.tyUILifterNomSpd.diMin;

	tyP1031MagSetTeach.tyMotionStdLifter.tyNumSlwSpd.diValueMax		:= p_tyNtParamCurr.tyUILifterSlwSpd.diMax;
	tyP1031MagSetTeach.tyMotionStdLifter.tyNumSlwSpd.diValueMin		:= p_tyNtParamCurr.tyUILifterSlwSpd.diMin;

END_ACTION
```

#### Act_Main_P1040.st
```iecst
ACTION Act_Main_P1040:

	//Display
	tyP1040ProdSet.tyProdSet.tyNumProdWidth.diValueMin		:= p_tyNtParamCurr.tyProdRcpWidth.diMin;
	tyP1040ProdSet.tyProdSet.tyNumProdWidth.diValueMax		:= p_tyNtParamCurr.tyProdRcpWidth.diMax;

	tyP1040ProdSet.tyProdSet.tyNumProdWidth2.diValueMin		:= p_tyNtParamCurr.tyProdRcpWidth.diMin;
	tyP1040ProdSet.tyProdSet.tyNumProdWidth2.diValueMax		:= p_tyNtParamCurr.tyProdRcpWidth.diMax;

	tyP1040ProdSet.tyProdSet.tyNumFirstSlt.diValueMin		:= p_tyNtParamCurr.diProjMagMinSlt;

	tyP1040ProdSet.tyProdSet.tyNumPitch.diValueMin			:= p_tyNtParamCurr.tyProdRcpPitch.diMin;

	tyP1040ProdSet.tyProdSet.tyNumProdWidthRear.diValueMin		:= p_tyNtParamCurr.tyProdRcpWidth.diMin;
	tyP1040ProdSet.tyProdSet.tyNumProdWidthRear.diValueMax		:= p_tyNtParamCurr.tyProdRcpWidth.diMax;
	tyP1040ProdSet.tyProdSet.tyNumPitchRear.diValueMin			:= p_tyNtParamCurr.tyProdRcpPitch.diMin;
	tyP1040ProdSet.tyProdSet.tyNumFirstSltRear.diValueMin		:= p_tyNtParamCurr.diProjMagMinSlt;

	tyP1040ProdSet.tyProdSet.tyDrpDnFlippedBrd.uiRtStat	:= TRUE;
	//Machine Mode
	IF p_tyNtParamCurr.bProjLaneBPrep THEN
		tyP1040ProdSet.tyProdSet.tyDrpDnMcMode.usiValueMaxIdx	:= 2;
		tyP1040ProdSet.tyProdSet.tyDrpDnMcMode.uiRtStat	:= FALSE;
	ELSE
		tyP1040ProdSet.tyProdSet.tyDrpDnMcMode.usiValueMaxIdx	:= 0;
		tyP1040ProdSet.tyProdSet.tyDrpDnMcMode.uiRtStat	:= TRUE;
	END_IF;

	//P1040 Product Settings
	FOR i := 1 TO c_uiP1040TableSize DO
		tyP1040ProdSet.tyProdSet.tyTableRecipe.a_tyStringDataCol0[i].sValue	:= UINT_TO_STRING(i);
		tyP1040ProdSet.tyProdSet.tyTableRecipe.a_tyStringDataCol1[i].sValue	:= p_tyProdRcpCurrList[i].sRcpNm;
		tyP1040ProdSet.tyProdSet.tyTableRecipe.a_tyStringDataCol2[i].sValue	:= p_tyProdRcpCurrList[i].sDisplayInfo;
	END_FOR

	tyP1040ProdSet.tyProdSet.tyBtnToptoBtm.bRtLk := FALSE;
	tyP1040ProdSet.tyProdSet.tyBtnToptoBtm.uiRtStat.0 := TRUE;

	IF p_tyNtParamCurr.bLFProdWidth2Prep THEN
		fUIInRtStatOff(ADR(tyP1040ProdSet.tyProdSet.tyNumProdWidth2.uiRtStat));
		fUIInRtStatHide(ADR(tyP1040ProdSet.tyProdSet.tyNumProdWidth.uiRtStat));

		tyP1040ProdSet.tyProdSet.tyTableRecipe.tyStringTitle2Col2Row0.sValue:= 'US | DS Width';
	ELSE
		fUIInRtStatHide(ADR(tyP1040ProdSet.tyProdSet.tyNumProdWidth2.uiRtStat));
		fUIInRtStatOff(ADR(tyP1040ProdSet.tyProdSet.tyNumProdWidth.uiRtStat));

		tyP1040ProdSet.tyProdSet.tyTableRecipe.tyStringTitle2Col2Row0.sValue:= 'Product Width';
	END_IF

	CASE p_tyNtParamCurr.eProjMag OF
		LDMagDual, LDMagTriple:
			fUIInRtStatOff(ADR(tyP1040ProdSet.tyProdSet.tyNotQuadrupleLyr.uiRtStat));
			fUIInRtStatHide(ADR(tyP1040ProdSet.tyProdSet.tyQuadrupleLyr.uiRtStat));

		LDMagQuadruple:
			fUIInRtStatHide(ADR(tyP1040ProdSet.tyProdSet.tyNotQuadrupleLyr.uiRtStat));
			fUIInRtStatOff(ADR(tyP1040ProdSet.tyProdSet.tyQuadrupleLyr.uiRtStat));
	END_CASE

	//Motorized Pusher
	tyP1040ProdSet.tyProdSet.tyNumMtrPshrExtSpd.diValueMin	:= p_tyNtParamCurr.tyProdRcpMtrPshrExtSpd.diMin;
	tyP1040ProdSet.tyProdSet.tyNumMtrPshrExtSpd.diValueMax	:= p_tyNtParamCurr.tyProdRcpMtrPshrExtSpd.diMax;

	tyP1040ProdSet.tyProdSet.tyNumMtrPshrExtTorq.diValueMin	:= p_tyNtParamCurr.tyProdRcpMtrPshrExtTorq.diMin;
	tyP1040ProdSet.tyProdSet.tyNumMtrPshrExtTorq.diValueMax	:= p_tyNtParamCurr.tyProdRcpMtrPshrExtTorq.diMax;

	tyP1040ProdSet.tyProdSet.tyNumMtrPshrExtSpd.uiRtStat.0	:= NOT p_tyNtParamCurr.bProjMotorizedPullerPrep;
	tyP1040ProdSet.tyProdSet.tyNumMtrPshrExtTorq.uiRtStat.0	:= NOT p_tyNtParamCurr.bProjMotorizedPullerPrep;

	tyP1040ProdSet.tyProdSet.tyNumPshrOffset.uiRtStat.0		:= NOT (p_tyNtParamCurr.bAWPusherPrep);
	tyP1040ProdSet.tyProdSet.tyTxtPshrOffset.uiRtStat.0		:= NOT (p_tyNtParamCurr.bAWPusherPrep);

END_ACTION
```

#### Act_Main_P1050.st
```iecst
ACTION Act_Main_P1050:

	//Display
	tyP1050LFSet.tyLdr.tyNumAfterOven.diValueMax	:= p_tyNtParamCurr.tyUILFIndexAfterOven.diMax;
	tyP1050LFSet.tyLdr.tyNumAfterOven.diValueMin	:= p_tyNtParamCurr.tyUILFIndexAfterOven.diMin;
	tyP1050LFSet.tyLdr.tyNumAfterOven2.diValueMax	:= p_tyNtParamCurr.tyUILFIndexAfterOven.diMax;
	tyP1050LFSet.tyLdr.tyNumAfterOven2.diValueMin	:= p_tyNtParamCurr.tyUILFIndexAfterOven.diMin;

	tyP1050LFSet.tyLdr.tyNumBeforeOven.diValueMax	:= p_tyNtParamCurr.tyUILFIndexBeforeOven.diMax;
	tyP1050LFSet.tyLdr.tyNumBeforeOven.diValueMin	:= p_tyNtParamCurr.tyUILFIndexBeforeOven.diMin;
	tyP1050LFSet.tyLdr.tyNumBeforeOven2.diValueMax	:= p_tyNtParamCurr.tyUILFIndexBeforeOven.diMax;
	tyP1050LFSet.tyLdr.tyNumBeforeOven2.diValueMin	:= p_tyNtParamCurr.tyUILFIndexBeforeOven.diMin;
	//Leader
	FOR i := 1 TO c_uiP1050TableSize DO
		tyP1050LFSet.tyLdr.tyTable1List.a_tyStringDataCol2[i].sValue	:= p_tyMcParamCurr.a_sLFIPAddr[i];
		tyP1050LFSet.tyLdr.tyTable1List.a_tyTxtDataCol3[i].usiValueIdx	:= (BOOL_TO_USINT(p_tyMcParamCurr.a_bLFOnline[i])) + 1;
	END_FOR

	//Parameter
	tyP1050LFSet.tyLdr.tyNumAfterOven.diValue	:= p_tyMcParamCurr.diLFMcIdxAfterOven;
	tyP1050LFSet.tyLdr.tyNumBeforeOven.diValue	:= p_tyMcParamCurr.diLFMcIdxBeforeOven;
	tyP1050LFSet.tyLdr.tyNumAfterOven2.diValue	:= p_tyMcParamCurr.diLFMcIdxAfterOven2;
	tyP1050LFSet.tyLdr.tyNumBeforeOven2.diValue	:= p_tyMcParamCurr.diLFMcIdxBeforeOven2;

END_ACTION
```

#### Act_Main_P1081.st
```iecst
ACTION Act_Main_P1081:

	//User Managment - User Access Right
	//Level 1
	IF p_tyUsrMgmtFullData.tyAccessRightLvl1.sNm <> '' THEN
		tyP1081UsrMgmtUsrAccessRgt.tyUsrAccessRgtLvl1.tyStringNm.sValue	:= p_tyUsrMgmtFullData.tyAccessRightLvl1.sNm;
		tyProperty.tyUITxtSnippets.sUsrMgmtUsrLv1Nm						:= p_tyUsrMgmtFullData.tyAccessRightLvl1.sNm;
	ELSE
		tyP1081UsrMgmtUsrAccessRgt.tyUsrAccessRgtLvl1.tyStringNm.sValue	:= tyProperty.tyUITxtSnippets.sUsrMgmtUsrLv1Nm;
	END_IF

	tyP1081UsrMgmtUsrAccessRgt.tyUsrAccessRgtLvl1.tyBtnOps.bValue		:= p_tyUsrMgmtFullData.tyAccessRightLvl1.bOpt;
	tyP1081UsrMgmtUsrAccessRgt.tyUsrAccessRgtLvl1.tyBtnProdSel.bValue	:= p_tyUsrMgmtFullData.tyAccessRightLvl1.bProdSel;
	tyP1081UsrMgmtUsrAccessRgt.tyUsrAccessRgtLvl1.tyBtnMagSel.bValue	:= p_tyUsrMgmtFullData.tyAccessRightLvl1.bMagSel;
	tyP1081UsrMgmtUsrAccessRgt.tyUsrAccessRgtLvl1.tyBtnMcInfo.bValue	:= p_tyUsrMgmtFullData.tyAccessRightLvl1.bMcInfo;
	tyP1081UsrMgmtUsrAccessRgt.tyUsrAccessRgtLvl1.tyBtnAlm.bValue		:= p_tyUsrMgmtFullData.tyAccessRightLvl1.bAlm;
	tyP1081UsrMgmtUsrAccessRgt.tyUsrAccessRgtLvl1.tyBtnBffrInfo.bValue	:= p_tyUsrMgmtFullData.tyAccessRightLvl1.bBffrInfo;
	tyP1081UsrMgmtUsrAccessRgt.tyUsrAccessRgtLvl1.tyBtnOvenInfo.bValue	:= p_tyUsrMgmtFullData.tyAccessRightLvl1.bOvenInfo;
	tyP1081UsrMgmtUsrAccessRgt.tyUsrAccessRgtLvl1.tyBtnMagInfo.bValue	:= p_tyUsrMgmtFullData.tyAccessRightLvl1.bMagInfo;
	tyP1081UsrMgmtUsrAccessRgt.tyUsrAccessRgtLvl1.tyBtnLFCtrl.bValue	:= p_tyUsrMgmtFullData.tyAccessRightLvl1.bLFCtrl;
	tyP1081UsrMgmtUsrAccessRgt.tyUsrAccessRgtLvl1.tyBtnManual.bValue	:= p_tyUsrMgmtFullData.tyAccessRightLvl1.bManual;
	tyP1081UsrMgmtUsrAccessRgt.tyUsrAccessRgtLvl1.tyBtnSimu.bValue		:= p_tyUsrMgmtFullData.tyAccessRightLvl1.bSimulation;
	tyP1081UsrMgmtUsrAccessRgt.tyUsrAccessRgtLvl1.tyBtnProdSet.bValue	:= p_tyUsrMgmtFullData.tyAccessRightLvl1.bProdSet;
	tyP1081UsrMgmtUsrAccessRgt.tyUsrAccessRgtLvl1.tyBtnMagSet.bValue	:= p_tyUsrMgmtFullData.tyAccessRightLvl1.bMagSet;
	tyP1081UsrMgmtUsrAccessRgt.tyUsrAccessRgtLvl1.tyBtnMcSet.bValue		:= p_tyUsrMgmtFullData.tyAccessRightLvl1.bMcSet;
	tyP1081UsrMgmtUsrAccessRgt.tyUsrAccessRgtLvl1.tyBtnLang.bValue		:= p_tyUsrMgmtFullData.tyAccessRightLvl1.bLang;
	tyP1081UsrMgmtUsrAccessRgt.tyUsrAccessRgtLvl1.tyBtnLFSet.bValue		:= p_tyUsrMgmtFullData.tyAccessRightLvl1.bLFSet;
	tyP1081UsrMgmtUsrAccessRgt.tyUsrAccessRgtLvl1.tyBtnChgParam.bValue	:= p_tyUsrMgmtFullData.tyAccessRightLvl1.bChgParam;

	//Level 2
	IF p_tyUsrMgmtFullData.tyAccessRightLvl2.sNm <> '' THEN
		tyP1081UsrMgmtUsrAccessRgt.tyUsrAccessRgtLvl2.tyStringNm.sValue	:= p_tyUsrMgmtFullData.tyAccessRightLvl2.sNm;
		tyProperty.tyUITxtSnippets.sUsrMgmtUsrLv2Nm						:= p_tyUsrMgmtFullData.tyAccessRightLvl2.sNm;
	ELSE
		tyP1081UsrMgmtUsrAccessRgt.tyUsrAccessRgtLvl2.tyStringNm.sValue	:= tyProperty.tyUITxtSnippets.sUsrMgmtUsrLv2Nm;
	END_IF

	tyP1081UsrMgmtUsrAccessRgt.tyUsrAccessRgtLvl2.tyBtnOps.bValue		:= p_tyUsrMgmtFullData.tyAccessRightLvl2.bOpt;
	tyP1081UsrMgmtUsrAccessRgt.tyUsrAccessRgtLvl2.tyBtnProdSel.bValue	:= p_tyUsrMgmtFullData.tyAccessRightLvl2.bProdSel;
	tyP1081UsrMgmtUsrAccessRgt.tyUsrAccessRgtLvl2.tyBtnMagSel.bValue	:= p_tyUsrMgmtFullData.tyAccessRightLvl2.bMagSel;
	tyP1081UsrMgmtUsrAccessRgt.tyUsrAccessRgtLvl2.tyBtnMcInfo.bValue	:= p_tyUsrMgmtFullData.tyAccessRightLvl2.bMcInfo;
	tyP1081UsrMgmtUsrAccessRgt.tyUsrAccessRgtLvl2.tyBtnAlm.bValue		:= p_tyUsrMgmtFullData.tyAccessRightLvl2.bAlm;
	tyP1081UsrMgmtUsrAccessRgt.tyUsrAccessRgtLvl2.tyBtnBffrInfo.bValue	:= p_tyUsrMgmtFullData.tyAccessRightLvl2.bBffrInfo;
	tyP1081UsrMgmtUsrAccessRgt.tyUsrAccessRgtLvl2.tyBtnOvenInfo.bValue	:= p_tyUsrMgmtFullData.tyAccessRightLvl2.bOvenInfo;
	tyP1081UsrMgmtUsrAccessRgt.tyUsrAccessRgtLvl2.tyBtnMagInfo.bValue	:= p_tyUsrMgmtFullData.tyAccessRightLvl2.bMagInfo;
	tyP1081UsrMgmtUsrAccessRgt.tyUsrAccessRgtLvl2.tyBtnLFCtrl.bValue	:= p_tyUsrMgmtFullData.tyAccessRightLvl2.bLFCtrl;
	tyP1081UsrMgmtUsrAccessRgt.tyUsrAccessRgtLvl2.tyBtnManual.bValue	:= p_tyUsrMgmtFullData.tyAccessRightLvl2.bManual;
	tyP1081UsrMgmtUsrAccessRgt.tyUsrAccessRgtLvl2.tyBtnSimu.bValue		:= p_tyUsrMgmtFullData.tyAccessRightLvl2.bSimulation;
	tyP1081UsrMgmtUsrAccessRgt.tyUsrAccessRgtLvl2.tyBtnProdSet.bValue	:= p_tyUsrMgmtFullData.tyAccessRightLvl2.bProdSet;
	tyP1081UsrMgmtUsrAccessRgt.tyUsrAccessRgtLvl2.tyBtnMagSet.bValue	:= p_tyUsrMgmtFullData.tyAccessRightLvl2.bMagSet;
	tyP1081UsrMgmtUsrAccessRgt.tyUsrAccessRgtLvl2.tyBtnMcSet.bValue		:= p_tyUsrMgmtFullData.tyAccessRightLvl2.bMcSet;
	tyP1081UsrMgmtUsrAccessRgt.tyUsrAccessRgtLvl2.tyBtnLang.bValue		:= p_tyUsrMgmtFullData.tyAccessRightLvl2.bLang;
	tyP1081UsrMgmtUsrAccessRgt.tyUsrAccessRgtLvl2.tyBtnLFSet.bValue		:= p_tyUsrMgmtFullData.tyAccessRightLvl2.bLFSet;
	tyP1081UsrMgmtUsrAccessRgt.tyUsrAccessRgtLvl2.tyBtnChgParam.bValue	:= p_tyUsrMgmtFullData.tyAccessRightLvl2.bChgParam;

	//Level 3
	IF p_tyUsrMgmtFullData.tyAccessRightLvl3.sNm <> '' THEN
		tyP1081UsrMgmtUsrAccessRgt.tyUsrAccessRgtLvl3.tyStringNm.sValue	:= p_tyUsrMgmtFullData.tyAccessRightLvl3.sNm;
		tyProperty.tyUITxtSnippets.sUsrMgmtUsrLv3Nm						:= p_tyUsrMgmtFullData.tyAccessRightLvl3.sNm;
	ELSE
		tyP1081UsrMgmtUsrAccessRgt.tyUsrAccessRgtLvl3.tyStringNm.sValue	:= tyProperty.tyUITxtSnippets.sUsrMgmtUsrLv3Nm;
	END_IF

	tyP1081UsrMgmtUsrAccessRgt.tyUsrAccessRgtLvl3.tyBtnOps.bValue		:= p_tyUsrMgmtFullData.tyAccessRightLvl3.bOpt;
	tyP1081UsrMgmtUsrAccessRgt.tyUsrAccessRgtLvl3.tyBtnProdSel.bValue	:= p_tyUsrMgmtFullData.tyAccessRightLvl3.bProdSel;
	tyP1081UsrMgmtUsrAccessRgt.tyUsrAccessRgtLvl3.tyBtnMagSel.bValue	:= p_tyUsrMgmtFullData.tyAccessRightLvl3.bMagSel;
	tyP1081UsrMgmtUsrAccessRgt.tyUsrAccessRgtLvl3.tyBtnMcInfo.bValue	:= p_tyUsrMgmtFullData.tyAccessRightLvl3.bMcInfo;
	tyP1081UsrMgmtUsrAccessRgt.tyUsrAccessRgtLvl3.tyBtnAlm.bValue		:= p_tyUsrMgmtFullData.tyAccessRightLvl3.bAlm;
	tyP1081UsrMgmtUsrAccessRgt.tyUsrAccessRgtLvl3.tyBtnBffrInfo.bValue	:= p_tyUsrMgmtFullData.tyAccessRightLvl3.bBffrInfo;
	tyP1081UsrMgmtUsrAccessRgt.tyUsrAccessRgtLvl3.tyBtnOvenInfo.bValue	:= p_tyUsrMgmtFullData.tyAccessRightLvl3.bOvenInfo;
	tyP1081UsrMgmtUsrAccessRgt.tyUsrAccessRgtLvl3.tyBtnMagInfo.bValue	:= p_tyUsrMgmtFullData.tyAccessRightLvl3.bMagInfo;
	tyP1081UsrMgmtUsrAccessRgt.tyUsrAccessRgtLvl3.tyBtnLFCtrl.bValue	:= p_tyUsrMgmtFullData.tyAccessRightLvl3.bLFCtrl;
	tyP1081UsrMgmtUsrAccessRgt.tyUsrAccessRgtLvl3.tyBtnManual.bValue	:= p_tyUsrMgmtFullData.tyAccessRightLvl3.bManual;
	tyP1081UsrMgmtUsrAccessRgt.tyUsrAccessRgtLvl3.tyBtnSimu.bValue		:= p_tyUsrMgmtFullData.tyAccessRightLvl3.bSimulation;
	tyP1081UsrMgmtUsrAccessRgt.tyUsrAccessRgtLvl3.tyBtnProdSet.bValue	:= p_tyUsrMgmtFullData.tyAccessRightLvl3.bProdSet;
	tyP1081UsrMgmtUsrAccessRgt.tyUsrAccessRgtLvl3.tyBtnMagSet.bValue	:= p_tyUsrMgmtFullData.tyAccessRightLvl3.bMagSet;
	tyP1081UsrMgmtUsrAccessRgt.tyUsrAccessRgtLvl3.tyBtnMcSet.bValue		:= p_tyUsrMgmtFullData.tyAccessRightLvl3.bMcSet;
	tyP1081UsrMgmtUsrAccessRgt.tyUsrAccessRgtLvl3.tyBtnLang.bValue		:= p_tyUsrMgmtFullData.tyAccessRightLvl3.bLang;
	tyP1081UsrMgmtUsrAccessRgt.tyUsrAccessRgtLvl3.tyBtnLFSet.bValue		:= p_tyUsrMgmtFullData.tyAccessRightLvl3.bLFSet;
	tyP1081UsrMgmtUsrAccessRgt.tyUsrAccessRgtLvl3.tyBtnChgParam.bValue	:= p_tyUsrMgmtFullData.tyAccessRightLvl3.bChgParam;

END_ACTION
```

#### Act_Main_P0003.st - not listed in the package file held
```iecst
ACTION Act_Main_P0003:

	tyP0003MMenu.tyMMenuGen.tyBitmapDSBIn.uiRtStat.0	:= TRUE;
	tyP0003MMenu.tyMMenuGen.tyBitmapDSBIn1.uiRtStat.0	:= TRUE;
	tyP0003MMenu.tyMMenuGen.tyBitmapDSBOut.uiRtStat.0	:= TRUE;
	tyP0003MMenu.tyMMenuGen.tyBitmapDSBOut1.uiRtStat.0	:= TRUE;
	tyP0003MMenu.tyMMenuGen.tyBitmapDSBComm.uiRtStat.0 := TRUE;
	tyP0003MMenu.tyMMenuGen.tyBitmapDSBComm.uiMaskRtStat.0 := TRUE;

////	FOR usidx := 1 TO SIZEOF(a_pBtn)/SIZEOF(a_pBtn[1]) DO
////		a_pBtn := ADR();
////	END_FOR

	//{TextSnippet_1} Position in Main Menu

	//hide corresponding button
//	tyP0003MMenu.tyMMenuBtn.tyBtnUnload.uiRtStat.0 :=  NOT p_tyNtParamCurr.bProjLifterMagPlatform;
//	tyP0003MMenu.tyMMenuBtn.tyBtnRlsNewMag1.uiRtStat.0 := p_tyNtParamCurr.bProjLifterMagPlatform;
//	tyP0003MMenu.tyMMenuBtn.tyBtnRlsNewMag2.uiRtStat.0 :=  p_tyNtParamCurr.bProjLifterMagPlatform;
//	tyP0003MMenu.tyMMenuBtn.tyBtnRlsNewMag3.uiRtStat.0 :=  p_tyNtParamCurr.bProjLifterMagPlatform;

END_ACTION
```

#### Package Logical/UI/UI/Act_Background - Change By Project

#### Act_ChgPage.st
```iecst
ACTION Act_ChgPage:

	(*Exit Page*)
	IF ((eChgPage <> eChgPageOld) OR (usiChgPage = 2)) AND p_bStartupRun = FALSE THEN

		usiChgPage	:= 2;

		CASE eChgPageOld OF

			UIP0700LFCtrl:
				Act_ExitP0700;

			UIP1000Lang:
				Act_ExitP1000;

			UIP1021McSetGen:
				Act_ExitP1021;

			UIP1022McSetVComm:
				Act_ExitP1022;

			UIP1023McSetHComm:
				Act_ExitP1023;

			UIP1024McSetAntiGap:
				Act_ExitP1024;

			UIP1025McSetAIVComm:
				Act_ExitP1025;

			UIP1026McSetTeach:
				Act_ExitP1026;

			UIP1027McSetUSBSet:
				Act_ExitP1027;

			UIP1028McSetRS232Set:
				Act_ExitP1028;

			UIP1031MagSetTeach:
				Act_ExitP1031;

			UIP1080UsrMgmt:
				Act_ExitP1080;

			UIP1081UsrMgmtUsrAccessRgt:
				Act_ExitP1081;

			ELSE
				usiChgPage	:= 1;

		END_CASE

		IF usiChgPage = 1 THEN
			eChgPageOld		:= eChgPage;
		END_IF

	(*Enter Page*)
	ELSIF usiChgPage = 1 THEN

		CASE eChgPage OF

			UIP0001Startup:
				Act_EntP0001Disp;

			UIP0002Menu:
				Act_EntP0002Disp;

			UIP0100Login:
				Act_EntP0100Disp;

			UIP0200OpsGen:
				Act_EntP0200Disp;

			UIP0201OpsTravLifter:
				Act_EntP0201Disp;

			UIP0202OpsMag1:
				Act_EntP0202Disp;

			UIP0203OpsMag2:
				Act_EntP0203Disp;

			UIP0204OpsMag3:
				Act_EntP0204Disp;

			UIP0205OpsAIV:
				Act_EntP0205Disp;

			UIP0206OpsMag4:
				Act_EntP0206Disp;

			UIP0300McInfo:
				Act_EntP0300Disp;

			UIP0400ProdSel:
				Act_EntP0400Disp;

			UIP0410MagSel:
				Act_EntP0410Disp;

			UIP0600Alm:
				Act_EntP0600Disp;

			UIP0700LFCtrl:
				Act_EntP0700Disp;

			UIP0800MagInfo:
				Act_EntP0800Disp;

			UIP0900GenIn:
				Act_EntP0900Disp;

			UIP0910GenOut:
				Act_EntP0910Disp;

			UIP0920MtrNPneuCtrl:
				Act_EntP0920Disp;

			UIP0921Shutter:
				Act_EntP0921Disp;

			UIP0923SafetyBar:
				Act_EntP0923Disp;

			UIP0924TrolleyLck:
				Act_EntP0924Disp;

			UIP0930MagConv1:
				Act_EntP0930Disp;

			UIP0931MagConv2:
				Act_EntP0931Disp;

			UIP0932MagConv3:
				Act_EntP0932Disp;

			UIP0933PullConv:
				Act_EntP0933Disp;

			UIP0934AW:
				Act_EntP0934Disp;

			UIP0935Lifter:
				Act_EntP0935Disp;

			UIP0936Trav:
				Act_EntP0936Disp;

			UIP0937AWPushOrPuller:
				Act_EntP0937Disp;

			UIP0939MagConv4:
				Act_EntP0939Disp;

			UIP0940CommCtrl:
				Act_EntP0940Disp;

			UIP0950Simu:
				Act_EntP0950Disp;

			UIP1000Lang:
				Act_EntP1000Disp;

			UIP1020McSetNavi:
				Act_EntP1020Disp;

			UIP1021McSetGen:
				Act_EntP1021Disp;

			UIP1022McSetVComm:
				Act_EntP1022Disp;

			UIP1023McSetHComm:
				Act_EntP1023Disp;

			UIP1024McSetAntiGap:
				Act_EntP1024Disp;

			UIP1025McSetAIVComm:
				Act_EntP1025Disp;

			UIP1026McSetTeach:
				Act_EntP1026Disp;

			UIP1027McSetUSBSet:
				Act_EntP1027Disp;

			UIP1028McSetRS232Set:
				Act_EntP1028Disp;

			UIP1030MagSet:
				Act_EntP1030Disp;

			UIP1031MagSetTeach:
				Act_EntP1031Disp;

			UIP1040ProdSet:
				Act_EntP1040Disp;

			UIP1050LFSet:
				Act_EntP1050Disp;

			UIP1080UsrMgmt:
				Act_EntP1080Disp;

			UIP1081UsrMgmtUsrAccessRgt:
				Act_EntP1081Disp;

		END_CASE

		usiChgPage	:= 0;

		tyProperty.tyVisu.uiChgPage	:= UDINT_TO_UINT(eChgPage);

	END_IF

END_ACTION
```

#### Act_OptPage.st
```iecst
ACTION Act_OptPage:

	//Prevent Screen Saver Interupt Program
	IF tyProperty.tyVisu.uiCurrPage <> 0 THEN
		eCurrPage := tyProperty.tyVisu.uiCurrPage;
	ELSE
		Act_OptP0000McStatus;
		Act_OptP0000RunningNm;
		Act_OptP0000StatDisp;
	END_IF

	Act_OptP0000DisableSSaver;
	Act_OptP0000TouchTimer;			//Auto Logout
	Act_OptP0000Hermes; //new for Hermes 1.3
	Act_OptP0002ToP1081UnlockCoverPB;

	IF (tyProperty.tyVisu.uiChgPage = 65535) AND (usiChgPage = 0) THEN

		Act_OptC0005GoHomeCtrl;
		Act_OptC0005ShowNotif;
		Act_OptC0005AutoCtrl;
		Act_OptC0005RstErr;
		Act_OptC0005StatBarCtrl;
		Act_OptC0005Buzzer;
		Act_OptC0005ChgPage;
		Act_OptC0007Notif;
		Act_OptC0009Info;

		Act_OptP0202InsertRmvMag;
		Act_OptP0203InsertRmvMag;
		Act_OptP0204InsertRmvMag;
		Act_OptP0200WorkOrderToLMC;

		CASE eCurrPage OF

			UIP0001Startup:
				Act_OptP0001Startup;

			UIP0100Login:
				Act_OptP0100Keypad;
				Act_OptP0100NomLogin;
				Act_OptP0100BypassLogin;
				Act_OptP0100Logout;

			UIP0200OpsGen:
				Act_OptP0200ChgPage;
				Act_OptP0200UpdtDat;
				Act_OptP0200VSMEMA;
				Act_OptP0200RcyMsg;
				Act_OptP0200ToP0204AccDat;
				Act_OptP0200ToP0204BypsInitConv;
				Act_OptP0202RstMnl;
				Act_OptP0203RstMnl;
				Act_OptP0204RstMnl;
				Act_OptP0200BarCodeScannerAndOthers;
				Act_OptP0200BarCodeChgRcp;
				Act_OptP0200Keypad;

			UIP0201OpsTravLifter:
				Act_OptP0201Navi;
				Act_OptP0201UpdtDat;
				Act_OptP0201IOMonitor;
				Act_OptP0201ChgParam;
				Act_OptP0200ToP0204AccDat;
				Act_OptP0200ToP0204BypsInitConv;
				Act_OptP0201CurrWorkOrderInfo; //new for Hermes 1.3
				Act_OptP0201QueryWorkOrderInfo; //new for Hermes 1.3
				Act_OptP0201QueryBoardInfo;//new for Hermes 1.3
				Act_OptP0201BarcodeScanner;//new for Hermes 1.3

			UIP0202OpsMag1:
				Act_OptP0202Navi;
				Act_OptP0202UpdtDat;
				Act_OptP0202IOMonitor;
				Act_OptP0202ChgPage;
				Act_OptP0202AIVDat;
				Act_OptP0202ChgParam;
				Act_OptP0200ToP0204AccDat;
				Act_OptP0200ToP0204BypsInitConv;
				Act_OptP0202ToP0204UnloadMag;

			UIP0203OpsMag2:
				Act_OptP0203Navi;
				Act_OptP0203UpdtDat;
				Act_OptP0203IOMonitor;
				Act_OptP0203ChgPage;
				Act_OptP0203AIVDat;
				Act_OptP0203ChgParam;
				Act_OptP0200ToP0204AccDat;
				Act_OptP0200ToP0204BypsInitConv;
				Act_OptP0202ToP0204UnloadMag;

			UIP0204OpsMag3:
				Act_OptP0204Navi;
				Act_OptP0204UpdtDat;
				Act_OptP0204IOMonitor;
				Act_OptP0204ChgPage;
				Act_OptP0204AIVDat;
				Act_OptP0204ChgParam;
				Act_OptP0200ToP0204AccDat;
				Act_OptP0200ToP0204BypsInitConv;
				Act_OptP0202ToP0204UnloadMag;

			UIP0205OpsAIV:
				Act_OptP0205Navi;
				Act_OptP0205IOMonitor;

			UIP0206OpsMag4:
				Act_OptP0206Navi;
				Act_OptP0206UpdtDat;
				Act_OptP0206IOMonitor;
				Act_OptP0206ChgPage;
				Act_OptP0206AIVDat;
				Act_OptP0206ChgParam;
				Act_OptP0200ToP0204AccDat;
				Act_OptP0200ToP0204BypsInitConv;
				Act_OptP0202ToP0204UnloadMag;

			UIP0300McInfo:

			UIP0400ProdSel:
				Act_OptP0400Search;
				Act_OptP0400Load;
				Act_OptP0400Preview;
				Act_OptP0400Table;
				Act_OptP0400Keypad;
				Act_OptP0400Mask;
				Act_OptP0400Sort;
				Act_OptP0400RcpPopUp;

			UIP0410MagSel:
				Act_OptP0410Navi;
				Act_OptP0410Load;
				Act_OptP0410Preview;
				Act_OptP0410Table;
				Act_OptP0410Mask;
				Act_OptP0410Sort;

			UIP0600Alm:
				Act_OptP0600Alm;
				Act_OptP0600RcyMsg;

			UIP0700LFCtrl:
				Act_OptP0700LFLeaderCtrl;
				Act_OptP0700Mask;
				Act_OptP0700Table;

			UIP0800MagInfo:
				Act_OptP0800Navi;
				Act_OptP0800Table1;
				Act_OptP0800Mag1Updt;
				Act_OptP0800Table2;
				Act_OptP0800Mag2Updt;
				Act_OptP0800Table3;
				Act_OptP0800Mag3Updt;
				Act_OptP0800Table4;
				Act_OptP0800Mag4Updt;

			UIP0002Menu, UIP0900GenIn, UIP0910GenOut, UIP0920MtrNPneuCtrl, UIP0921Shutter, UIP0923SafetyBar, UIP0924TrolleyLck, UIP0930MagConv1, UIP0931MagConv2, UIP0932MagConv3, UIP0933PullConv, UIP0934AW, UIP0935Lifter, UIP0936Trav, UIP0937AWPushOrPuller, UIP0939MagConv4, UIP0940CommCtrl:
				IF eCurrPage = UIP0002Menu THEN
					Act_OptP0002Mask;
					Act_OptP0002ChgPage;
					Act_OptP0002MsgGuide;
					Act_OptP0002UpdtData;
				END_IF

				Act_OptP0002ManualCtrl;
				Act_OptP0910RstMnl;
				Act_OptP0921RstMnl;
				Act_OptP0923RstMnl;
				Act_OptP0924RstMnl;
				Act_OptP0930RstMnl;
				Act_OptP0931RstMnl;
				Act_OptP0932RstMnl;
				Act_OptP0933RstMnl;
				Act_OptP0934RstMnl;
				Act_OptP0935RstMnl;
				Act_OptP0936RstMnl;
				Act_OptP0937RstMnl;
				Act_OptP0939RstMnl;
				Act_OptP0940RstMnl;
				Act_OptP0950RstMnl;
				Act_OptP0202RstMnl;
				Act_OptP0203RstMnl;
				Act_OptP0204RstMnl;
				Act_OptP0205RstMnl;
				Act_OptP0206RstMnl;

				IF bUIManualMod = TRUE THEN

					//General Input
					Act_OptP0900ReadDI;

					//General Output
					Act_OptP0910WriteDO;

					//MtrNPneuCtrl
					Act_OptP0920FullMask;
					Act_OptP0920ChgPage;

					//Inlet & Outlet Shutter
					Act_OptP0921DualMask;
					Act_OptP0921Navi;
					Act_OptP0921InletShutterChgLyr; //inlet shutter
					Act_OptP0921InletShutterSen;
					Act_OptP0921InletShutterFB;
					Act_OptP0921InletShutterFBStat;
					Act_OptP0921InletShutterDC;
					Act_OptP0921InletShutterChgLyr2;
					Act_OptP0921InletShutterSen2;
					Act_OptP0921InletShutterFB2;
					Act_OptP0921InletShutterFBStat2;
					Act_OptP0921InletShutterDC2;
					Act_OptP0921InletShutterChgLyr3;
					Act_OptP0921InletShutterSen3;
					Act_OptP0921InletShutterFB3;
					Act_OptP0921InletShutterFBStat3;
					Act_OptP0921InletShutterDC3;
					Act_OptP0921OutletShutterChgLyr; //outlet shutter
					Act_OptP0921OutletShutterSen;
					Act_OptP0921OutletShutterFB;
					Act_OptP0921OutletShutterFBStat;
					Act_OptP0921OutletShutterDC;
					Act_OptP0921OutletShutterChgLyr2;
					Act_OptP0921OutletShutterSen2;
					Act_OptP0921OutletShutterFB2;
					Act_OptP0921OutletShutterFBStat2;
					Act_OptP0921OutletShutterDC2;

					//Safety Bar
					Act_OptP0923DualMask;
					Act_OptP0923Navi;
					Act_OptP0923Mag1SafetyBarChgLyr;
					Act_OptP0923Mag1SafetyBarSen;
					Act_OptP0923Mag1SafetyBarFB;
					Act_OptP0923Mag1SafetyBarFBStat;
					Act_OptP0923Mag1SafetyBarDC;
					Act_OptP0923Mag2SafetyBarChgLyr;
					Act_OptP0923Mag2SafetyBarSen;
					Act_OptP0923Mag2SafetyBarFB;
					Act_OptP0923Mag2SafetyBarFBStat;
					Act_OptP0923Mag2SafetyBarDC;
					Act_OptP0923Mag3SafetyBarChgLyr;
					Act_OptP0923Mag3SafetyBarSen;
					Act_OptP0923Mag3SafetyBarFB;
					Act_OptP0923Mag3SafetyBarFBStat;
					Act_OptP0923Mag3SafetyBarDC;

					//Trolley lock
					Act_OptP0924FullMask;
					Act_OptP0924Navi;
					Act_OptP0924TrolleyLckChgLyr;
					Act_OptP0924TrolleyLckSen;
					Act_OptP0924TrolleyLckFB;
					Act_OptP0924TrolleyLckFBStat;
					Act_OptP0924TrolleyLckDC;

					//Magazine Conveyor 1
					Act_OptP0930FullMask;
					Act_OptP0930Navi;
					Act_OptP0930MagConv1ChgLyr;
					Act_OptP0930MagConv1Sen;
					Act_OptP0930MagConv1FB;
					Act_OptP0930MagConv1FBStat;
					Act_OptP0930MagConv1DC;

					//Magazine Conveyor 2
					Act_OptP0931FullMask;
					Act_OptP0931Navi;
					Act_OptP0931MagConv2ChgLyr;
					Act_OptP0931MagConv2Sen;
					Act_OptP0931MagConv2FB;
					Act_OptP0931MagConv2FBStat;
					Act_OptP0931MagConv2DC;

					//Magazine Conveyor 3
					Act_OptP0932FullMask;
					Act_OptP0932Navi;
					Act_OptP0932MagConv3ChgLyr;
					Act_OptP0932MagConv3Sen;
					Act_OptP0932MagConv3FB;
					Act_OptP0932MagConv3FBStat;
					Act_OptP0932MagConv3DC;

					//Puller Conveyor
					Act_OptP0933FullMask;
					Act_OptP0933Navi;
					Act_OptP0933PullerConvChgLyr;
					Act_OptP0933PullerConvSen;
					Act_OptP0933PullerConvFB;
					Act_OptP0933PullerConvFBStat;
					Act_OptP0933PullerConvDC;
					Act_OptP0933Keypad;
					//AutoWidth
					Act_OptP0934FullMask;
					Act_OptP0934Navi;
					Act_OptP0934FBCtrl;
					Act_OptP0934FBStat;
					Act_OptP0934Mask;
					Act_OptP0934UpdtDat;
					Act_OptP0934Keypad;

					//Lifter
					Act_OptP0935FullMask;
					Act_OptP0935Navi;
					Act_OptP0935FBCtrl;
					Act_OptP0935FBStat;
					Act_OptP0935Mask;
					Act_OptP0935UpdtDat;
					Act_OptP0935Keypad;

					//Traverser
					Act_OptP0936FullMask;
					Act_OptP0936Navi;
					Act_OptP0936FBCtrl;
					Act_OptP0936FBStat;
					Act_OptP0936Mask;
					Act_OptP0936UpdtDat;
					Act_OptP0936Keypad;

					//Pusher Or Puller Auto Width
					Act_OptP0937FullMask;
					Act_OptP0937Navi;
					Act_OptP0937FBCtrl;
					Act_OptP0937FBStat;
					Act_OptP0937Mask;
					Act_OptP0937UpdtDat;
					Act_OptP0937Keypad;

					//Magazine Conveyor 4
					Act_OptP0939FullMask;
					Act_OptP0939Navi;
					Act_OptP0939MagConv4ChgLyr;
					Act_OptP0939MagConv4Sen;
					Act_OptP0939MagConv4FB;
					Act_OptP0939MagConv4FBStat;
					Act_OptP0939MagConv4DC;

					//Communication
					Act_OptP0940FullMask;
					Act_OptP0940ReadDI;
					Act_OptP0940WriteDO;

				END_IF

			UIP0950Simu:
				Act_OptP0950Ctrl;
				Act_OptP0950SimuMod;

			UIP1000Lang:
				Act_OptP1000SelectLang;
				Act_OptP1000Keypad;

			UIP1020McSetNavi:
				Act_OptP1020Navi;

			UIP1021McSetGen:
				Act_OptP1021Navi;
				Act_OptP1021Save;
				Act_OptP1021Keypad;
				Act_OptP1021Teach;
				Act_OptP1021IPAddr;
				Act_OptP1021SubnetMask;
				Act_OptP1021DHCPSetting;

			UIP1022McSetVComm:
				Act_OptP1022Navi;
				Act_OptP1022Save;
				Act_OptP1022DisLF;
				Act_OptP1022Keypad; //new for Hermes 1.3

			UIP1023McSetHComm:
				Act_OptP1023Navi;
				Act_OptP1023ShowLyr;
				Act_OptP1023Save;
				Act_OptP1023DSSel;
				Act_OptP1023Keypad;

			UIP1024McSetAntiGap:
				Act_OptP1024Navi;
				Act_OptP1024Save;
				Act_OptP1024Keypad;

//			UIP1025McSetAIVComm:
//				Act_OptP1025Navi;
//				Act_OptP1025Save;
//				Act_OptP1025Keypad;

			UIP1026McSetTeach:
				Act_OptP1026Navi;
				Act_OptP1026FullMask;
				Act_OptP1026Mnl;

				//Traverser
				Act_OptP1026TravTeach;
				Act_OptP1026TravFBCtrl;
				Act_OptP1026TravFBStat;
				Act_OptP1026TravMask;
				Act_OptP1026TravUpdtDat;
				Act_OptP1026TravKeypad;
				Act_OptP1026TravRstMnl;

				//Lifter
				Act_OptP1026LifterTeach;
				Act_OptP1026LifterFBCtrl;
				Act_OptP1026LifterFBStat;
				Act_OptP1026LifterMask;
				Act_OptP1026LifterUpdtDat;
				Act_OptP1026LifterKeypad;
				Act_OptP1026LifterRstMnl;

			UIP1027McSetUSBSet:
				Act_OptP1027Navi;
				Act_OptP1027Save;
				Act_OptP1027Keypad;

			UIP1028McSetRS232Set:
				Act_OptP1028Navi;
				Act_OptP1028Save;
				Act_OptP1028Keypad;

			UIP1030MagSet:
				Act_OptP1030Mask;
				Act_OptP1030Save;
				Act_OptP1030Del;
				Act_OptP1030Table;
				Act_OptP1030LoadData;
				Act_OptP1030Keypad;
				Act_OptP1030Teach;
				Act_OptP1030Sort;

			UIP1031MagSetTeach:
				Act_OptP1031Navi;
				Act_OptP1031FullMask;
				Act_OptP1031Mnl;

				//Traverser
				Act_OptP1031TravTeach;
				Act_OptP1031TravFBCtrl;
				Act_OptP1031TravFBStat;
				Act_OptP1031TravMask;
				Act_OptP1031TravUpdtDat;
				Act_OptP1031TravKeypad;
				Act_OptP1031TravRstMnl;

				//Lifter
				Act_OptP1031LifterTeach;
				Act_OptP1031LifterFBCtrl;
				Act_OptP1031LifterFBStat;
				Act_OptP1031LifterMask;
				Act_OptP1031LifterUpdtDat;
				Act_OptP1031LifterKeypad;
				Act_OptP1031LifterRstMnl;

			UIP1040ProdSet:
				Act_OptP1040Mask;
				Act_OptP1040Save;
				Act_OptP1040Del;
				Act_OptP1040Table;
				Act_OptP1040LoadData;
				Act_OptP1040Search;
				Act_OptP1040Keypad;
				Act_OptP1040Limit;
				Act_OptP1040ToXML;
				Act_OptP1040FromXML;
				Act_OptP1040Sort;
				Act_OptP1040RcpPopUp;

			UIP1050LFSet:
				Act_OptP1050Keypad;
				Act_OptP1050Edit;
				Act_OptP1050Online;
				Act_OptP1050Offline;
				Act_OptP1050Delete;
				Act_OptP1050ShftUp;
				Act_OptP1050ShftDwn;
				Act_OptP1050Mask;
				Act_OptP1050Table;
				Act_OptP1050Oven;

			UIP1080UsrMgmt:
				Act_OptP1080Keypad;
				Act_OptP1080AddUsr;
				Act_OptP1080DelUsr;
				Act_OptP1080EditUsr;
				Act_OptP1080EditAccess;
				Act_OptP1080Table;

			UIP1081UsrMgmtUsrAccessRgt:
				Act_OptP1081Navi;
				Act_OptP1081Save;
				Act_OptP1081Load;
				Act_OptP1081Keypad;

		END_CASE

	END_IF

END_ACTION
```

#### Act_OptC0005AutoCtrl.st
```iecst
ACTION Act_OptC0005AutoCtrl:

	//Control
	//Error
	IF EDGEPOS(p_bAlarmErr = TRUE AND p_bOpsStatusStop = FALSE) THEN

		tyCommon.tyMain.tyBtnStart.bRtCompl	:= FALSE;
		tyCommon.tyMain.tyBtnStop.bRtCompl	:= FALSE;
		tyCommon.tyMain.tyBtnStep.bRtCompl	:= FALSE;

		tyCommon.tyMain.tyBtnStart.bValue	:= FALSE;
		tyCommon.tyMain.tyBtnStop.bValue	:= FALSE;
		tyCommon.tyMain.tyBtnStep.bValue	:= FALSE;

		eOpsAct	:= OperationsActError;

	ELSE

		IF p_eOpsStat = OperationsActError AND p_eOpsStatus = Done THEN
			eOpsAct	:= OperationsActIdle;
		END_IF

	END_IF

	//Start
	IF tyCommon.tyMain.tyBtnStart.bRtCompl = TRUE THEN

		IF tyCommon.tyMain.tyBtnStart.bValue = TRUE THEN

			IF eCurrPage <> UIP0200OpsGen AND eCurrPage <> UIP0201OpsTravLifter AND eCurrPage <> UIP0202OpsMag1 AND eCurrPage <> UIP0203OpsMag2 AND eCurrPage <> UIP0204OpsMag3 THEN

				IF bChgPage = FALSE THEN
					bChgPage	:= TRUE;
					eChgPage	:= UIP0200OpsGen;
				ELSE
					IF eChgPage <> UIP0200OpsGen THEN
						bChgPage	:= FALSE;

						tyCommon.tyMain.tyBtnStart.bRtCompl	:= FALSE;
						tyCommon.tyMain.tyBtnStart.bValue	:= FALSE;
					END_IF
				END_IF

			ELSE
				bChgPage	:= FALSE;

				tyCommon.tyMain.tyBtnStart.bValue	:= FALSE;

				tyCommon.tyMain.tyBtnStop.bRtCompl	:= FALSE;
				tyCommon.tyMain.tyBtnStep.bRtCompl	:= FALSE;

				tyCommon.tyMain.tyBtnStop.bValue	:= FALSE;
				tyCommon.tyMain.tyBtnStep.bValue	:= FALSE;
			END_IF

		ELSE

			eOpsAct	:= OperationsActStart;

			IF p_eOpsStat = OperationsActStart AND p_eOpsStatus = Done THEN
				eOpsAct	:= OperationsActIdle;

				tyCommon.tyMain.tyBtnStart.bRtCompl	:= FALSE;
			END_IF

		END_IF

	END_IF

	//Stop
	IF tyCommon.tyMain.tyBtnStop.bRtCompl = TRUE THEN

		IF tyCommon.tyMain.tyBtnStop.bValue = TRUE THEN

			tyCommon.tyMain.tyBtnStop.bValue	:= FALSE;

			tyCommon.tyMain.tyBtnStart.bRtCompl	:= FALSE;
			tyCommon.tyMain.tyBtnStep.bRtCompl	:= FALSE;

			tyCommon.tyMain.tyBtnStart.bValue	:= FALSE;
			tyCommon.tyMain.tyBtnStep.bValue	:= FALSE;

		ELSE

			eOpsAct	:= OperationsActStop;

			IF p_eOpsStat = OperationsActStop AND p_eOpsStatus = Done THEN
				eOpsAct	:= OperationsActIdle;

				tyCommon.tyMain.tyBtnStop.bRtCompl	:= FALSE;
			END_IF

		END_IF

	END_IF

	//Step
	IF tyCommon.tyMain.tyBtnStep.bRtCompl = TRUE THEN

		IF tyCommon.tyMain.tyBtnStep.bValue = TRUE THEN

			IF eCurrPage <> UIP0200OpsGen AND eCurrPage <> UIP0201OpsTravLifter AND eCurrPage <> UIP0202OpsMag1 AND eCurrPage <> UIP0203OpsMag2 AND eCurrPage <> UIP0204OpsMag3 THEN

				IF bChgPage = FALSE THEN
					bChgPage	:= TRUE;
					eChgPage	:= UIP0200OpsGen;
				ELSE
					IF eChgPage <> UIP0200OpsGen THEN
						bChgPage	:= FALSE;

						tyCommon.tyMain.tyBtnStep.bRtCompl	:= FALSE;
						tyCommon.tyMain.tyBtnStep.bValue	:= FALSE;
					END_IF
				END_IF

			ELSE
				bChgPage	:= FALSE;

				tyCommon.tyMain.tyBtnStep.bValue	:= FALSE;

				tyCommon.tyMain.tyBtnStart.bRtCompl	:= FALSE;
				tyCommon.tyMain.tyBtnStop.bRtCompl	:= FALSE;

				tyCommon.tyMain.tyBtnStart.bValue	:= FALSE;
				tyCommon.tyMain.tyBtnStop.bValue	:= FALSE;
			END_IF

		ELSE

			eOpsAct	:= OperationsActStep;

			IF p_eOpsStat = OperationsActStep AND p_eOpsStatus = Done THEN
				eOpsAct	:= OperationsActIdle;

				tyCommon.tyMain.tyBtnStep.bRtCompl	:= FALSE;
			END_IF

		END_IF

	END_IF

	//Display
	//Auto Step
	IF p_tyMcParamCurr.bAutoStepEn = TRUE THEN
		fUIInRtStatOff(ADR(tyCommon.tyMain.tyBtnStep.uiRtStat));
	ELSE
		fUIInRtStatHide(ADR(tyCommon.tyMain.tyBtnStep.uiRtStat));
		fUIInRtStatHide(ADR(tyCommon.tyMain.tyBtnStep.uiMaskRtStat));
	END_IF

	//Mask
	IF (p_bAlarmErr = TRUE) OR (bUIManualMod = TRUE) OR (p_tyDI.bSafetyRlySig = FALSE) OR (tyCommon.tyMain.tyBtnHome.uiMaskRtStat.0 = FALSE) OR eCurrPage = UIP0950Simu THEN
		fUIInRtStatOff(ADR(tyCommon.tyMain.tyBtnStart.uiMaskRtStat));
		fUIInRtStatOff(ADR(tyCommon.tyMain.tyBtnStop.uiMaskRtStat));

		IF p_tyMcParamCurr.bAutoStepEn = TRUE THEN
			fUIInRtStatOff(ADR(tyCommon.tyMain.tyBtnStep.uiMaskRtStat));
		END_IF

	ELSE

		IF p_eOpsOpsStatus = OperationsStatusRun THEN

			fUIInRtStatOff(ADR(tyCommon.tyMain.tyBtnStart.uiMaskRtStat));
			fUIInRtStatHide(ADR(tyCommon.tyMain.tyBtnStop.uiMaskRtStat));
			fUIInRtStatHide(ADR(tyCommon.tyMain.tyBtnStep.uiMaskRtStat));

		ELSIF p_eOpsOpsStatus = OperationsStatusCycleStopping THEN

			fUIInRtStatHide(ADR(tyCommon.tyMain.tyBtnStart.uiMaskRtStat));
			fUIInRtStatOff(ADR(tyCommon.tyMain.tyBtnStop.uiMaskRtStat));
			fUIInRtStatHide(ADR(tyCommon.tyMain.tyBtnStep.uiMaskRtStat));

		ELSIF p_eOpsOpsStatus = OperationsStatusStep THEN

			fUIInRtStatHide(ADR(tyCommon.tyMain.tyBtnStart.uiMaskRtStat));
			fUIInRtStatHide(ADR(tyCommon.tyMain.tyBtnStop.uiMaskRtStat));

			IF p_eOpsStatus = Busy THEN
				fUIInRtStatOff(ADR(tyCommon.tyMain.tyBtnStep.uiMaskRtStat));
			ELSE
				fUIInRtStatHide(ADR(tyCommon.tyMain.tyBtnStep.uiMaskRtStat));
			END_IF

		ELSE

			fUIInRtStatHide(ADR(tyCommon.tyMain.tyBtnStart.uiMaskRtStat));
			fUIInRtStatOff(ADR(tyCommon.tyMain.tyBtnStop.uiMaskRtStat));
			fUIInRtStatHide(ADR(tyCommon.tyMain.tyBtnStep.uiMaskRtStat));

		END_IF

	END_IF

END_ACTION
```

#### Act_OptC0005Buzzer.st
```iecst
ACTION Act_OptC0005Buzzer:

	IF tyCommon.tyMain.tyBtnBuzzer.bRtCompl = TRUE THEN
		tyCommon.tyMain.tyBtnBuzzer.bRtCompl	:= FALSE;

		IF tyCommon.tyMain.tyBtnBuzzer.bValue = TRUE THEN
			tyCommon.tyMain.tyBtnBuzzer.usiBitmapIdx	:= 2;

			bMuteBuz	:= TRUE;
		ELSE
			tyCommon.tyMain.tyBtnBuzzer.usiBitmapIdx	:= 1;

			bMuteBuz	:= FALSE;
		END_IF

	END_IF

	//Mute Buzzer
	IF EDGEPOS((p_bAlarmErr OR p_bAlarmWarning OR p_bAlarmInfo) (*AND NOT bUIManualMod*)) THEN

		tyCommon.tyMain.tyBtnBuzzer.bValue				:= FALSE;
		tyCommon.tyMain.tyBtnBuzzer.bRtLk				:= FALSE;
		tyCommon.tyMain.tyBtnBuzzer.usiBitmapIdx		:= 1;

		bMuteBuz	:= FALSE;

	ELSIF (p_bAlarmErr OR p_bAlarmWarning OR p_bAlarmInfo) THEN

		IF p_bAlarmInfoLF AND NOT (p_bAlarmErr OR p_bAlarmWarning OR (p_bAlarmInfo AND NOT p_bAlarmInfoLF)) THEN

			IF p_tyMcParamCurr.bLFBuzMute THEN

				tyCommon.tyMain.tyBtnBuzzer.bValue				:= FALSE;
				tyCommon.tyMain.tyBtnBuzzer.bRtLk				:= TRUE;
				tyCommon.tyMain.tyBtnBuzzer.usiBitmapIdx		:= 0;

				bMuteBuz	:= FALSE;
			ELSE
				tyCommon.tyMain.tyBtnBuzzer.bRtLk				:= FALSE;

				IF tyCommon.tyMain.tyBtnBuzzer.bValue THEN
					tyCommon.tyMain.tyBtnBuzzer.usiBitmapIdx		:= 2;
				ELSE
					tyCommon.tyMain.tyBtnBuzzer.usiBitmapIdx		:= 1;
				END_IF

			END_IF
		ELSE

			tyCommon.tyMain.tyBtnBuzzer.bRtLk				:= FALSE;

			IF tyCommon.tyMain.tyBtnBuzzer.bValue THEN
				tyCommon.tyMain.tyBtnBuzzer.usiBitmapIdx		:= 2;
			ELSE
				tyCommon.tyMain.tyBtnBuzzer.usiBitmapIdx		:= 1;
			END_IF
		END_IF

	ELSIF NOT(p_bAlarmErr OR p_bAlarmWarning OR p_bAlarmInfo) (*OR bUIManualMod*) THEN
		tyCommon.tyMain.tyBtnBuzzer.bRtLk				:= TRUE;
		tyCommon.tyMain.tyBtnBuzzer.usiBitmapIdx		:= 0;

		bMuteBuz	:= FALSE;
	END_IF

END_ACTION
```

#### Act_OptC0005ChgPage.st
```iecst
ACTION Act_OptC0005ChgPage:

	//Control Alarm and Warning
	IF tyCommon.tyMain.tyBtnAlarm.bRtCompl = TRUE THEN
		tyCommon.tyMain.tyBtnAlarm.bRtCompl := FALSE;
		IF p_bAlarmErr = TRUE OR p_bAlarmWarning THEN
			eChgPage  := UIP0600Alm;
		END_IF
	END_IF

	//Display Alarm Button Control
//	tyCommon.tyMain.tyBtnAlarm.uiRtStat.0		:= NOT (p_bAlarmErr OR p_bAlarmWarning) ;
	tyCommon.tyMain.tyHotspotNaviStart.uiRtStat.0 := tyCommon.tyMain.tyBtnStart.uiMaskRtStat.0;
	//Mask Control
//	tyCommon.tyMain.tyBtnAlarm.uiMaskRtStat.0	:= NOT ((p_bAlarmErr OR p_bAlarmWarning) AND (eCurrPage = UIP0600Alm));

	IF tyCommon.tyMain.tyHotspotNaviStart.bRtCompl = TRUE THEN
		tyCommon.tyMain.tyHotspotNaviStart.bRtCompl := FALSE;

		IF p_bAlarmErr = TRUE OR p_bAlarmWarning THEN
			eChgPage	:= UIP0600Alm;
		END_IF
	END_IF

END_ACTION
```

#### Act_OptC0005GoHomeCtrl.st
```iecst
ACTION Act_OptC0005GoHomeCtrl:

	//Control
	IF tyCommon.tyMain.tyBtnHome.bRtCompl = TRUE THEN
		tyCommon.tyMain.tyBtnHome.bRtCompl	:= FALSE;
		eChgPage							:= UIP0002Menu;
	END_IF

	//Mask
	IF tyP0100Login.tyLogin.tyBtnLogin.bRtCompl						OR tyP0100Login.tyLogout.tyBtnLogout.bRtCompl
		OR tyP0400ProdSel.tyProdSel.tyBtnLoad.bRtCompl				OR tyP0400ProdSel.tyProdSel.tyStringSearch.bRtCompl
		OR tyP0410MagSel.tyMagSel.tyBtnLoad.bRtCompl				OR tyP0800MagInfo.tyMagInfo1.tyBtnMag1SetEmpty.bRtCompl
		OR tyP0800MagInfo.tyMagInfo1.tyBtnMag2SetEmpty.bRtCompl		OR tyP0800MagInfo.tyMagInfo2.tyBtnMag3SetEmpty.bRtCompl
		OR tyP1030MagSet.tyMagSet.tyBtnDelete.bRtCompl				OR tyP1030MagSet.tyMagSet.tyBtnSave.bRtCompl
		OR tyP1040ProdSet.tyProdSet.tyBtnDelete.bRtCompl			OR tyP1040ProdSet.tyProdSet.tyBtnSave.bRtCompl
		OR tyP1040ProdSet.tyProdSet.tyBtnToXML.bRtCompl				OR tyP1040ProdSet.tyProdSet.tyBtnFromXML.bRtCompl
		OR tyP1050LFSet.tyLdr.tyBtnDelete.bRtCompl					OR tyP1050LFSet.tyLdr.tyBtnOnline.bRtCompl
		OR tyP1050LFSet.tyLdr.tyBtnOffline.bRtCompl					OR tyP1050LFSet.tyLdr.tyBtnShftUp.bRtCompl
		OR tyP1050LFSet.tyLdr.tyBtnShftDwn.bRtCompl					OR tyP1080UsrMgmt.tyUsrMgmt.tyBtnDeleteUsr.bRtCompl
		OR tyP1080UsrMgmt.tyUsrMgmt.tyBtnEditDetail.bRtCompl		OR tyP1080UsrMgmt.tyUsrMgmt.tyBtnNewUsr.bRtCompl
		OR tyCommon.tySet.tyBtnSave.bRtCompl						OR bTeachTravPosA
		OR bTeachTravPosB											OR bTeachTravPosMag1
		OR bTeachTravPosMag2										OR bTeachTravPosMag3
		OR bTeachTravPosMag4
		OR bTeachLifterPosA											OR bTeachLifterPosB
		OR bTeachLifterMag1Slt1Pos									OR bTeachLifterMag2Slt1Pos
		OR bTeachLifterMag3Slt1Pos 									OR bTeachLifterMag4Slt1Pos
		OR p_bSimuStatusRun
		THEN

		fUIInRtStatOff(ADR(tyCommon.tyMain.tyBtnHome.uiMaskRtStat));

	ELSIF bUIManualMod THEN
		fUIInRtStatHide(ADR(tyCommon.tyMain.tyBtnHome.uiMaskRtStat));

	ELSE
		fUIInRtStatHide(ADR(tyCommon.tyMain.tyBtnHome.uiMaskRtStat));

	END_IF

END_ACTION
```

#### Act_OptC0005RstErr.st
```iecst
ACTION Act_OptC0005RstErr:

	//Control
	IF tyCommon.tyMain.tyBtnReset.bRtCompl = TRUE THEN
		eRstErrAct	:= RstErrActRun;
		IF NOT p_tyDI.bCurtainSafetySig2 THEN
			bSafetyCurtainReset := TRUE;//Curtain reset button
		END_IF

//		fbCurtainRstDly(IN:= TRUE);

		IF p_eRstErrStat = RstErrActRun AND p_eRstErrStatus =  Done THEN
			eRstErrAct	:= RstErrActIdle;
			tyCommon.tyMain.tyBtnReset.bRtCompl	:= FALSE;
		END_IF

	END_IF

	//Mask
	IF p_bAlarmErr = TRUE OR p_bAlarmWarning = TRUE OR p_tyDI.bSafetyRlySig = FALSE THEN
		fUIInRtStatHide(ADR(tyCommon.tyMain.tyBtnReset.uiMaskRtStat));
	ELSE
		fUIInRtStatOff(ADR(tyCommon.tyMain.tyBtnReset.uiMaskRtStat));
	END_IF

	//Curtain Reset delay
//	fbCurtainRstDly;
//	IF fbCurtainRstDly.Q AND bSafetyCurtainReset THEN
//		IF (p_eRstErrStat = RstErrActRun AND p_eRstErrStatus =  Done) OR p_eRstErrStat = RstErrActIdle THEN
//			fbCurtainRstDly(IN:= FALSE);
//			bSafetyCurtainReset := FALSE;
//		END_IF
//	END_IF
	IF bSafetyCurtainReset THEN
		fbCurtainRstDly(IN:=TRUE);

		IF fbCurtainRstDly.Q THEN
			fbCurtainRstDly(IN:= FALSE);
			bSafetyCurtainReset := FALSE;
		END_IF
	END_IF
END_ACTION
```

#### Act_OptC0005ShowNotif.st
```iecst
ACTION Act_OptC0005ShowNotif:

	//Control
	IF tyCommon.tyMain.tyBtnNotification.bRtCompl = TRUE THEN
		tyCommon.tyMain.tyBtnNotification.bRtCompl		:= FALSE;

		fUIInRtStatOff(ADR(tyCommon.tyNotif.tyLyr.uiRtStat));
	END_IF

END_ACTION
```

#### Act_OptC0005StatBarCtrl.st
```iecst
ACTION Act_OptC0005StatBarCtrl:

	//Error / Warning / Info
	IF p_bAlarmErr = TRUE OR p_bAlarmWarning = TRUE OR p_bAlarmInfo = TRUE THEN

		fbErrBlinkTm(IN := TRUE);
		IF fbErrBlinkTm.Q = TRUE THEN
			fbErrBlinkTm(IN := FALSE);

			IF p_bAlarmErr = TRUE THEN

				IF tyCommon.tyMain.tyBitmapStatBar.usiValueIdx = 1 THEN
					tyCommon.tyMain.tyBitmapStatBar.usiValueIdx	:= 0;
				ELSE
					tyCommon.tyMain.tyBitmapStatBar.usiValueIdx	:= 1;
				END_IF

			ELSE

				IF tyCommon.tyMain.tyBitmapStatBar.usiValueIdx = 3 THEN
					tyCommon.tyMain.tyBitmapStatBar.usiValueIdx	:= 0;
				ELSE
					tyCommon.tyMain.tyBitmapStatBar.usiValueIdx	:= 3;
				END_IF

			END_IF

		END_IF

	//Safety Relay Signal Activated
	ELSIF p_tyDI.bSafetyRlySig = FALSE THEN

		fbRstBlinkTm(IN := TRUE);
		IF fbRstBlinkTm.Q = TRUE THEN
			fbRstBlinkTm(IN := FALSE);

			IF tyCommon.tyMain.tyBitmapStatBar.usiValueIdx = 5 THEN
				tyCommon.tyMain.tyBitmapStatBar.usiValueIdx	:= 6;
			ELSE
				tyCommon.tyMain.tyBitmapStatBar.usiValueIdx	:= 5;
			END_IF

		END_IF

	//Manual Running
	ELSIF bUIManualMod THEN
		tyCommon.tyMain.tyBitmapStatBar.usiValueIdx	:= 0;

	//Operation Cycle Stopping
	ELSIF p_eOpsOpsStatus = OperationsStatusCycleStopping OR p_eSimuSimuStatus = SimulationsStatusCycleStopping  THEN

		fbStopBlinkTm(IN := TRUE);
		IF fbStopBlinkTm.Q = TRUE THEN
			fbStopBlinkTm(IN := FALSE);

			IF tyCommon.tyMain.tyBitmapStatBar.usiValueIdx = 1 THEN
				tyCommon.tyMain.tyBitmapStatBar.usiValueIdx	:= 2;
			ELSE
				tyCommon.tyMain.tyBitmapStatBar.usiValueIdx	:= 1;
			END_IF

		END_IF

	//Operation Stepping
	ELSIF p_eOpsOpsStatus = OperationsStatusStep THEN
		tyCommon.tyMain.tyBitmapStatBar.usiValueIdx	:= 3;

	//Operation Running
	ELSIF p_eOpsOpsStatus = OperationsStatusRun OR p_eSimuSimuStatus = SimulationsStatusRun THEN
		tyCommon.tyMain.tyBitmapStatBar.usiValueIdx	:= 2;

	//Standby
	ELSE
		tyCommon.tyMain.tyBitmapStatBar.usiValueIdx	:= 0;

	END_IF

END_ACTION
```

#### Act_OptC0007Notif.st
```iecst
ACTION Act_OptC0007Notif:

	//Display
	//User Level
	tyCommon.tyNotif.tyTxtUsrLv.usiValueIdx	:= UDINT_TO_USINT(p_tyUsrMgmtCurrUsr.eUsrLvl);
	tyCommon.tyNotif.tyStringUsrNm.sValue	:= p_tyUsrMgmtCurrUsr.sUsrNm;
	tyCommon.tyNotif.tyTxtLFMc.uiRtStat.0	:= NOT (p_tyNtParamCurr.bLFPrep AND p_tyMcParamCurr.bLFEn);

	IF p_tyNtParamCurr.bLFUsrSetPrep = TRUE THEN
		IF p_tyMcParamCurr.bLFLeaderMc = TRUE THEN
			tyCommon.tyNotif.tyTxtLFMc.usiValueIdx		:= 0;
		ELSE
			IF p_tyMcParamCurr.bSectionLeader = TRUE THEN
				tyCommon.tyNotif.tyTxtLFMc.usiValueIdx		:= 2;
			ELSE
				tyCommon.tyNotif.tyTxtLFMc.usiValueIdx		:= 1;
			END_IF
		END_IF
	END_IF

	//Show Info
	tyCommon.tyNotif.tyBitmapShowInfo.uiRtStat.0	:= p_bAlarmInfo = FALSE;
	tyCommon.tyNotif.tyHotspotShowInfo.uiRtStat.0	:= p_bAlarmInfo = FALSE;

	//Control
	IF tyCommon.tyNotif.tyLyr.uiRtStat.0 = FALSE THEN

		IF tyCommon.tyNotif.tyHotspotClose.bRtCompl = TRUE THEN
			tyCommon.tyNotif.tyHotspotClose.bRtCompl	:= FALSE;

			fUIInRtStatHide(ADR(tyCommon.tyNotif.tyLyr.uiRtStat));

		ELSIF tyCommon.tyNotif.tyHotspotShowInfo.bRtCompl = TRUE THEN
			tyCommon.tyNotif.tyHotspotShowInfo.bRtCompl	:= FALSE;

			fUIInRtStatOff(ADR(tyCommon.tyInfo.tyLyr.uiRtStat));
			fUIInRtStatHide(ADR(tyCommon.tyNotif.tyLyr.uiRtStat));

		END_IF

	END_IF

END_ACTION
```

#### Act_EntP0000Disp.st
```iecst
ACTION Act_EntP0000Disp:

	//Access Address
	p_tyP0000SSaver ACCESS ADR(tyP0000SSaver.tySSaver);
	p_tyC0008MsgBox ACCESS ADR(tyP0000SSaver.tyMsgBoxHide);
END_ACTION
```

#### Act_OptP0000Hermes.st
```iecst
ACTION Act_OptP0000Hermes: //Can receive at anytime, at any Page

	//SendBordInfo can be received at anytime, at any Page
	IF (p_bRcvBoardInfoIncompl AND tyCommon.tyInfo.tyHotspotClose.bRtCompl = TRUE) OR EDGENEG (p_bRcvBoardInfoOk) OR tyP0201OpsTravLifter.tyQueryBoardInfo.tyBtnQueryBoardInfo.bValue = FALSE THEN //Reset
		bQueryBoardInfo := FALSE;
		tyP0201OpsTravLifter.tyQueryBoardInfo.tyBtnQueryBoardInfo.bValue := FALSE;
	END_IF

	//Reset QueryWorkOrderInfo when Close C0009 Info
	IF EDGEPOS (tyCommon.tyInfo.tyHotspotClose.bRtCompl = TRUE OR tyP0201OpsTravLifter.tyCurrWorkOrderInfo.tyBtnQueryWorkOrderInfo.bValue = FALSE OR p_bRcvWorkOrderInfo1) THEN
		bQueryWorkOrderInfo := FALSE;
		tyP0201OpsTravLifter.tyCurrWorkOrderInfo.tyBtnQueryWorkOrderInfo.bValue := FALSE;
	END_IF

	//Configure update can happen at anytime, at any Page (Can modify to Reset this when User Press tyCommon.tyInfo.tyHotspotClose.bRtCompl)
	IF p_bRmtUpdateUIData = TRUE OR p_bSvyUpdateUIData = TRUE THEN

		//Update UI Upstream Configure
//		tyP1023McSetHComm.tyUSHermes.tyNumSndAliveTm.diValue		:= TIME_TO_DINT(p_tyHermesConfiguration.a_tyUSParam[0].tSndAlive);
//		tyP1023McSetHComm.tyUSHermes.tyNumLaneID.diValue			:= INT_TO_DINT(p_tyHermesConfiguration.a_tyUSParam[0].iLaneID);
//		tyP1023McSetHComm.tyUSHermes.tyNumHostPort.diValue			:= UINT_TO_DINT(p_tyHermesConfiguration.a_tyUSParam[0].uiHostPort);
//		tyP1023McSetHComm.tyUSHermes.tyStringHostAddr.sValue		:= p_tyHermesConfiguration.a_tyUSParam[0].sHostAddress;
//		tyP1023McSetHComm.tyUSHermes.tyBtnCheckAliveResponse.bValue	:= p_tyHermesConfiguration.a_tyUSParam[0].bFeatureCheckAliveResponse;
//		tyP1023McSetHComm.tyUSHermes.tyBtnCmpTypeId.bValue			:= p_tyHermesConfiguration.a_tyUSParam[0].bCmpTypeId;
//		tyP1023McSetHComm.tyUSHermes.tyBtnCmpParam.bValue			:= p_tyHermesConfiguration.a_tyUSParam[0].bCmpParam;
//		tyP1023McSetHComm.tyUSHermes.tyBtnOverWrite.bValue			:= p_tyHermesConfiguration.a_tyUSParam[0].bOverwrite;
//		tyP1023McSetHComm.tyUSHermes.tyBtnBoardForecast.bValue		:= p_tyHermesConfiguration.a_tyUSParam[0].bFeatureBoardForecast;//new
//		tyP1023McSetHComm.tyUSHermes.tyBtnQueryBoardInfo.bValue		:= p_tyHermesConfiguration.a_tyUSParam[0].bFeatureQueryBoardInfo;//new

		//Update UI Downstream Configure
		tyP1023McSetHComm.tyDSHermesA.tyNumSndAliveTm.diValue		:= TIME_TO_DINT(p_tyHermesConfiguration.a_tyDSParam[0].tSndAlive);
		tyP1023McSetHComm.tyDSHermesA.tyNumSvrPort.diValue			:= UINT_TO_DINT(p_tyHermesConfiguration.a_tyDSParam[0].uiSvrPort);
		tyP1023McSetHComm.tyDSHermesA.tyNumLaneID.diValue			:= INT_TO_DINT(p_tyHermesConfiguration.a_tyDSParam[0].iLaneID);
		tyP1023McSetHComm.tyDSHermesA.tyBtnCheckAliveResponse.bValue	:= p_tyHermesConfiguration.a_tyDSParam[0].bFeatureCheckAliveResponse;
		tyP1023McSetHComm.tyDSHermesA.tyBtnBoardForecast.bValue	    := p_tyHermesConfiguration.a_tyDSParam[0].bFeatureBoardForecast;//new
		tyP1023McSetHComm.tyDSHermesA.tyBtnSendBoardInfo.bValue	    := p_tyHermesConfiguration.a_tyDSParam[0].bFeatureSendBoardInfo;//new

		//Update UI Supervisory Configure
		tyP1022McSetVComm.tyVComSvy.tyNumSndAliveTm.diValue	    	:= TIME_TO_DINT(p_tyHermesConfiguration.tySvyParam.tSndAlive);
		tyP1022McSetVComm.tyVComSvy.tyNumSvySystemPort.diValue	    := UINT_TO_DINT(p_tyHermesConfiguration.tySvyParam.uiSvySvstemPort);
		tyP1022McSetVComm.tyVComSvy.tyBtnConfiguration.bValue		:= p_tyHermesConfiguration.tySvyParam.bFeatureConfiguration;
		tyP1022McSetVComm.tyVComSvy.tyBtnCheckAliveResponse.bValue	:= p_tyHermesConfiguration.tySvyParam.bFeatureCheckAliveResponse;
		tyP1022McSetVComm.tyVComSvy.tyBtnBoardTracking.bValue		:= p_tyHermesConfiguration.tySvyParam.bFeatureBoardTracking;
		tyP1022McSetVComm.tyVComSvy.tyBtnQueryWorkOrderInfo.bValue	:= p_tyHermesConfiguration.tySvyParam.bFeatureQueryWorkOrderInfo;
		tyP1022McSetVComm.tyVComSvy.tyBtnSendWorkOrderInfo.bValue   := p_tyHermesConfiguration.tySvyParam.bFeatureSendWorkOrderInfo;

		//Update UI Mc Name and Backup Mc Name of P1021
		tyP1021McSetGen.tyGen.tyStringMcNm.sValue			    	:= p_tyMcParamCurr.sMcNm; //String[30] doesnt tally with MachineId String[80] currently.
		tyP1021McSetGen.tyGenBkUp.tyStringMcNm	                    := tyP1021McSetGen.tyGen.tyStringMcNm;

		//Update Backup Param P1022
		tyP1022McSetVComm.tyVComSelBkUp	    := tyP1022McSetVComm.tyVComSel;
		tyP1022McSetVComm.tyVComSvyBkUp	    := tyP1022McSetVComm.tyVComSvy;
		tyP1022McSetVComm.tyLFBkUp		    := tyP1022McSetVComm.tyLF;

		//Update Backup Param P1023
//		tyP1023McSetHComm.tyUSSelBkUp		:= tyP1023McSetHComm.tyUSSel;
//		tyP1023McSetHComm.tyUSSMEMABkUp		:= tyP1023McSetHComm.tyUSSMEMA;
//		tyP1023McSetHComm.tyUSHermesBkUp	:= tyP1023McSetHComm.tyUSHermes;
		tyP1023McSetHComm.tyDSSelABkUp		:= tyP1023McSetHComm.tyDSSelA;
		tyP1023McSetHComm.tyDSSMEMAABkUp		:= tyP1023McSetHComm.tyDSSMEMAA;
		tyP1023McSetHComm.tyDSHermesABkUp	:= tyP1023McSetHComm.tyDSHermesA;

	END_IF

END_ACTION
```

#### Act_OptP0000TouchTimer.st
```iecst
ACTION Act_OptP0000TouchTimer:

	IF bLoginSuccess AND p_tyNtParamCurr.bAutoLogoutPrep AND p_tyMcParamCurr.bAutoLogoutEn THEN

		fbTouchTm();

		fbAutoLogoutTm(IN:= NOT fbTouchTm.bPressed, PT:=DINT_TO_TIME(p_tyMcParamCurr.diAutoLogoutTmInSec));

		//Reset Time When Pressed
		IF fbTouchTm.bPressed THEN
			fbAutoLogoutTm(IN:=FALSE);
		END_IF

		//Auto Logout
		IF fbAutoLogoutTm.Q THEN

			bPromptSessionExp	:= TRUE;
			p_tyC0008MsgBox ACCESS ADR(tyP0000SSaver.tyMsgBoxLoginAsk);

			IF bChgPageDone=FALSE THEN

				IF eCurrPage<>UIP0002Menu THEN
					CASE eCurrPage OF

						UIP0900GenIn, UIP0910GenOut, UIP0920MtrNPneuCtrl,UIP0921Shutter, UIP0930MagConv1, UIP0931MagConv2, UIP0932MagConv3, UIP0933PullConv, UIP0934AW, UIP0935Lifter, UIP0936Trav, UIP0939MagConv4, UIP0940CommCtrl, UIP0950Simu:

							eChgPage		:= UIP0002Menu;

							tyP0002Menu.tyMenu.tyBtnMnlRst.bRtCompl := TRUE ;

							bChgPageDone	:= TRUE;

						UIP1000Lang, UIP1021McSetGen, UIP1022McSetVComm, UIP1023McSetHComm, UIP1024McSetAntiGap, UIP1025McSetAIVComm, UIP1026McSetTeach, UIP1030MagSet, UIP1031MagSetTeach,UIP1040ProdSet, UIP1050LFSet, UIP1080UsrMgmt, UIP1081UsrMgmtUsrAccessRgt:

							IF tyCommon.tySet.tyBtnSave.uiMaskRtStat.0 = FALSE THEN

								eChgPage	:= UIP0002Menu;

								bChgPageDone	:= TRUE;

							ELSE

								eChgPage		:= UIP0002Menu;

								IF eCurrPage= UIP1021McSetGen THEN

									tyP1021McSetGen.tyMsgBoxExitAsk.tyBtnYes.bRtCompl := TRUE;

									bChgPageDone	:= TRUE;

								ELSIF eCurrPage= UIP1022McSetVComm THEN

									tyP1022McSetVComm.tyMsgBoxExitAsk.tyBtnYes.bRtCompl := TRUE;

									bChgPageDone	:= TRUE;

								ELSIF eCurrPage= UIP1023McSetHComm THEN

									tyP1023McSetHComm.tyMsgBoxExitAsk.tyBtnYes.bRtCompl := TRUE;

									bChgPageDone	:= TRUE;

								ELSIF eCurrPage= UIP1024McSetAntiGap THEN

									tyP1024McSetAntiGap.tyMsgBoxExitAsk.tyBtnYes.bRtCompl := TRUE;

									bChgPageDone	:= TRUE;

								ELSIF eCurrPage= UIP1026McSetTeach THEN

									tyP1026McSetTeach.tyMsgBoxExitAsk.tyBtnYes.bRtCompl := TRUE;

									bChgPageDone	:= TRUE;

								ELSIF eCurrPage= UIP1030MagSet THEN

									tyP1030MagSet.tyMsgBoxExitAsk.tyBtnYes.bRtCompl := TRUE;

									bChgPageDone	:= TRUE;

								ELSIF eCurrPage= UIP1031MagSetTeach THEN

									tyP1031MagSetTeach.tyMsgBoxExitAsk.tyBtnYes.bRtCompl := TRUE;

									bChgPageDone	:= TRUE;

								ELSE  //language page
									bChgPageDone	:= TRUE;
								END_IF

							END_IF

						ELSE
							eChgPage		:= UIP0002Menu;

							bChgPageDone	:= TRUE;

					END_CASE

				ELSE
					bChgPageDone	:= TRUE;
				END_IF

			END_IF

			IF bChgPageDone THEN

				eUsrMgmtAct	:= UsrMgmtActLogout;

				IF p_eUsrMgmtStat = UsrMgmtActLogout AND p_eUsrMgmtStatus = Done THEN
					eUsrMgmtAct	:= UsrMgmtActIdle;

					bLoginSuccess	:= FALSE;

					bChgPageDone	:= FALSE;

					fbAutoLogoutTm(IN:=FALSE);

				END_IF

			END_IF

		END_IF

	ELSE
		fbAutoLogoutTm(IN:=FALSE);
		bChgPageDone	:= FALSE;
	END_IF

	//Prompt Relogin After Auto Logout
	IF tyP0000SSaver.tyMsgBoxLoginAsk.tyBtnYes.bRtCompl = TRUE THEN
		tyP0000SSaver.tyMsgBoxLoginAsk.tyBtnYes.bRtCompl 	:= FALSE;
		tyP0000SSaver.tyMsgBoxLoginAsk.tyBtnYes.bValue		:= FALSE;
		p_tyC0008MsgBox ACCESS ADR(tyP0000SSaver.tyMsgBoxHide);
		bPromptSessionExp :=FALSE;

	ELSIF tyP0000SSaver.tyMsgBoxLoginAsk.tyBtnNo.bRtCompl = TRUE THEN
		tyP0000SSaver.tyMsgBoxLoginAsk.tyBtnNo.bRtCompl 	:= FALSE;
		tyP0000SSaver.tyMsgBoxLoginAsk.tyBtnNo.bValue		:= FALSE;
		p_tyC0008MsgBox ACCESS ADR(tyP0000SSaver.tyMsgBoxHide);
		eChgPage		:= UIP0100Login;
		bPromptSessionExp :=FALSE;
	END_IF

END_ACTION
```

#### Act_EntP0001Disp.st
```iecst
ACTION Act_EntP0001Disp:

	//UI Property Access
	p_tyVisu ACCESS ADR(tyProperty.tyVisu);

	p_tyKeypad ACCESS ADR(tyProperty.tyKeypad);

	p_tyTxtSnippets ACCESS ADR(tyProperty.tyUITxtSnippets);

	p_tyC0008MsgBox ACCESS ADR(tyP0001Startup.tyMsgBoxHide);

	//Access Address
	p_tyP0001Startup ACCESS ADR(tyP0001Startup.tyStartup);

	p_tyP0001Initial ACCESS ADR(tyP0001Startup.tyInitial);

	fUIInRtStatHide(ADR(tyP0001Startup.tyInitial.tyLyr.uiRtStat));

END_ACTION
```
